C03652=1220.015,344.206,-72.673,-176.049,7.398,148.250
C03653=1220.012,344.454,-72.705,-176.047,7.400,148.250
C03654=1220.007,344.702,-72.737,-176.045,7.403,148.251
C03655=1220.003,344.950,-72.769,-176.043,7.406,148.251
C03656=1219.998,345.198,-72.801,-176.042,7.408,148.251
C03657=1219.994,345.445,-72.833,-176.040,7.412,148.251
C03658=1219.990,345.693,-72.864,-176.038,7.414,148.251
C03659=1219.986,345.942,-72.897,-176.036,7.418,148.252
C03660=1219.982,346.189,-72.928,-176.034,7.420,148.252
C03661=1219.977,346.437,-72.961,-176.032,7.423,148.252
C03662=1219.974,346.685,-72.993,-176.030,7.426,148.252
C03663=1219.969,346.932,-73.025,-176.028,7.428,148.252
C03664=1219.965,347.180,-73.057,-176.027,7.431,148.252
C03665=1219.961,347.429,-73.089,-176.024,7.434,148.253
C03666=1219.956,347.676,-73.121,-176.023,7.437,148.253
C03667=1219.953,347.924,-73.153,-176.021,7.439,148.253
C03668=1219.948,348.173,-73.186,-176.019,7.443,148.253
C03669=1219.945,348.421,-73.217,-176.017,7.445,148.253
C03670=1219.940,348.668,-73.250,-176.015,7.448,148.254
C03671=1219.936,348.916,-73.282,-176.013,7.451,148.254
C03672=1219.932,349.164,-73.314,-176.012,7.453,148.254
C03673=1219.928,349.412,-73.346,-176.010,7.457,148.254
C03674=1219.923,349.660,-73.378,-176.008,7.459,148.254
C03675=1219.919,349.907,-73.411,-176.006,7.462,148.255
C03676=1219.915,350.155,-73.443,-176.004,7.465,148.255
C03677=1219.911,350.403,-73.475,-176.003,7.468,148.255
C03678=1219.906,350.651,-73.507,-176.001,7.471,148.255
C03679=1219.902,350.899,-73.540,-175.999,7.474,148.256
C03680=1219.898,351.147,-73.572,-175.997,7.476,148.256
C03681=1219.894,351.395,-73.605,-175.996,7.479,148.256
C03682=1219.890,351.642,-73.637,-175.994,7.482,148.256
C03683=1219.886,351.890,-73.669,-175.992,7.485,148.256
C03684=1219.882,352.138,-73.701,-175.990,7.488,148.257
C03685=1219.878,352.386,-73.734,-175.988,7.491,148.257
C03686=1219.873,352.634,-73.767,-175.987,7.493,148.257
C03687=1219.869,352.882,-73.798,-175.985,7.497,148.257
C03688=1219.865,353.130,-73.831,-175.983,7.499,148.258
C03689=1219.861,353.378,-73.863,-175.982,7.502,148.258
C03690=1219.857,353.626,-73.896,-175.979,7.505,148.258
C03691=1219.853,353.874,-73.929,-175.978,7.508,148.258
C03692=1219.848,354.121,-73.960,-175.976,7.510,148.258
C03693=1219.844,354.369,-73.993,-175.974,7.514,148.259
C03694=1219.840,354.617,-74.026,-175.973,7.517,148.259
C03695=1219.836,354.864,-74.059,-175.971,7.519,148.259
C03696=1219.832,355.113,-74.091,-175.969,7.522,148.259
C03697=1219.827,355.360,-74.124,-175.967,7.525,148.260
C03698=1219.823,355.608,-74.156,-175.966,7.528,148.260
C03699=1219.819,355.856,-74.188,-175.964,7.530,148.260
C03700=1219.815,356.104,-74.221,-175.962,7.534,148.260
C03701=1219.811,356.352,-74.253,-175.961,7.536,148.261
C03702=1219.807,356.600,-74.286,-175.959,7.539,148.261
C03703=1219.803,356.847,-74.319,-175.957,7.542,148.261
C03704=1219.798,357.095,-74.351,-175.956,7.545,148.261
C03705=1219.794,357.343,-74.384,-175.954,7.547,148.262
C03706=1219.790,357.591,-74.416,-175.952,7.551,148.262
C03707=1219.786,357.839,-74.450,-175.951,7.554,148.262
C03708=1219.782,358.087,-74.481,-175.949,7.556,148.262
C03709=1219.778,358.334,-74.515,-175.948,7.559,148.263
C03710=1219.774,358.582,-74.548,-175.946,7.562,148.263
C03711=1219.769,358.830,-74.580,-175.944,7.565,148.263
C03712=1219.766,359.078,-74.613,-175.943,7.568,148.264
C03713=1219.761,359.326,-74.645,-175.941,7.571,148.264
C03714=1219.757,359.573,-74.678,-175.939,7.574,148.264
C03715=1219.753,359.821,-74.711,-175.938,7.576,148.264
C03716=1219.749,360.069,-74.743,-175.936,7.579,148.265
C03717=1219.745,360.317,-74.776,-175.934,7.582,148.265
C03718=1219.741,360.564,-74.809,-175.933,7.585,148.265
C03719=1219.736,360.813,-74.842,-175.931,7.588,148.265
C03720=1219.732,361.061,-74.875,-175.930,7.590,148.266
C03721=1219.729,361.308,-74.907,-175.928,7.594,148.266
C03722=1219.725,361.556,-74.941,-175.926,7.596,148.266
C03723=1219.720,361.804,-74.973,-175.925,7.599,148.267
C03724=1219.716,362.052,-75.006,-175.923,7.602,148.267
C03725=1219.712,362.300,-75.039,-175.922,7.605,148.267
C03726=1219.708,362.547,-75.072,-175.920,7.608,148.267
C03727=1219.704,362.795,-75.104,-175.919,7.611,148.268
C03728=1219.699,363.042,-75.137,-175.917,7.613,148.268
C03729=1219.695,363.290,-75.170,-175.915,7.617,148.268
C03730=1219.691,363.538,-75.203,-175.914,7.619,148.269
C03731=1219.687,363.785,-75.237,-175.913,7.622,148.269
C03732=1219.682,364.034,-75.269,-175.911,7.625,148.269
C03733=1219.678,364.282,-75.302,-175.909,7.628,148.270
C03734=1219.674,364.529,-75.335,-175.908,7.631,148.270
C03735=1219.670,364.777,-75.368,-175.906,7.634,148.270
C03736=1219.667,365.024,-75.401,-175.905,7.636,148.270
C03737=1219.662,365.272,-75.434,-175.904,7.639,148.271
C03738=1219.658,365.521,-75.467,-175.902,7.643,148.271
C03739=1219.654,365.768,-75.500,-175.900,7.645,148.271
C03740=1219.650,366.016,-75.533,-175.899,7.648,148.272
C03741=1219.646,366.264,-75.566,-175.897,7.651,148.272
C03742=1219.641,366.511,-75.599,-175.896,7.653,148.272
C03743=1219.637,366.791,-75.637,-175.894,7.657,148.273
C03744=1219.633,367.072,-75.674,-175.893,7.660,148.273
C03745=1219.628,367.352,-75.712,-175.891,7.663,148.274
C03746=1219.623,367.631,-75.749,-175.889,7.667,148.274
C03747=1219.619,367.879,-75.782,-175.888,7.670,148.274
C03748=1219.615,368.127,-75.815,-175.887,7.672,148.275
C03749=1219.611,368.374,-75.849,-175.885,7.675,148.275
C03750=1219.607,368.622,-75.882,-175.884,7.678,148.275
C03751=1219.603,368.870,-75.915,-175.883,7.680,148.276
C03752=1219.598,369.117,-75.948,-175.881,7.683,148.276
C03753=1219.594,369.365,-75.981,-175.880,7.686,148.276
C03754=1219.590,369.613,-76.014,-175.878,7.690,148.277
C03755=1219.586,369.861,-76.047,-175.877,7.692,148.277
C03756=1219.582,370.108,-76.081,-175.876,7.695,148.277
C03757=1219.578,370.356,-76.114,-175.874,7.698,148.278
C03758=1219.574,370.604,-76.147,-175.873,7.701,148.278
C03759=1219.569,370.853,-76.181,-175.872,7.703,148.278
C03760=1219.565,371.100,-76.214,-175.870,7.706,148.279
C03761=1219.561,371.348,-76.247,-175.869,7.709,148.279
C03762=1219.557,371.595,-76.281,-175.868,7.712,148.279
C03763=1219.553,371.843,-76.314,-175.867,7.714,148.280
C03764=1219.549,372.091,-76.348,-175.865,7.717,148.280
C03765=1219.545,372.338,-76.381,-175.864,7.720,148.280
C03766=1219.541,372.586,-76.414,-175.863,7.723,148.281
C03767=1219.537,372.834,-76.447,-175.861,7.726,148.281
C03768=1219.532,373.082,-76.480,-175.860,7.729,148.282
C03769=1219.529,373.329,-76.514,-175.859,7.732,148.282
C03770=1219.524,373.577,-76.548,-175.857,7.734,148.282
C03771=1219.520,373.825,-76.581,-175.856,7.737,148.283
C03772=1219.516,374.073,-76.614,-175.855,7.740,148.283
C03773=1219.512,374.321,-76.648,-175.854,7.743,148.283
C03774=1219.508,374.568,-76.681,-175.852,7.746,148.284
C03775=1219.504,374.815,-76.715,-175.851,7.748,148.284
C03776=1219.500,375.063,-76.748,-175.850,7.751,148.285
C03777=1219.495,375.311,-76.782,-175.849,7.754,148.285
C03778=1219.492,375.559,-76.816,-175.848,7.757,148.285
C03779=1219.488,375.807,-76.849,-175.846,7.760,148.286
C03780=1219.483,376.054,-76.882,-175.845,7.763,148.286
C03781=1219.479,376.302,-76.915,-175.844,7.765,148.287
C03782=1219.475,376.549,-76.949,-175.843,7.767,148.287
C03783=1219.471,376.797,-76.983,-175.842,7.770,148.287
C03784=1219.466,377.045,-77.016,-175.841,7.773,148.288
C03785=1219.463,377.293,-77.050,-175.840,7.776,148.288
C03786=1219.459,377.541,-77.083,-175.839,7.779,148.289
C03787=1219.454,377.789,-77.117,-175.838,7.781,148.289
C03788=1219.450,378.036,-77.151,-175.836,7.784,148.289
C03789=1219.446,378.283,-77.184,-175.835,7.787,148.290
C03790=1219.442,378.531,-77.217,-175.834,7.790,148.290
C03791=1219.439,378.779,-77.252,-175.833,7.793,148.291
C03792=1219.434,379.027,-77.285,-175.832,7.796,148.291
C03793=1219.430,379.274,-77.319,-175.830,7.798,148.291
C03794=1219.426,379.522,-77.352,-175.830,7.800,148.292
C03795=1219.422,379.770,-77.386,-175.829,7.803,148.292
C03796=1219.417,380.017,-77.420,-175.827,7.806,148.292
C03797=1219.414,380.265,-77.454,-175.826,7.809,148.293
C03798=1219.410,380.513,-77.487,-175.825,7.812,148.293
C03799=1219.405,380.761,-77.521,-175.824,7.814,148.294
C03800=1219.401,381.008,-77.554,-175.823,7.817,148.294
C03801=1219.397,381.255,-77.588,-175.823,7.820,148.295
C03802=1219.394,381.504,-77.622,-175.821,7.822,148.295
C03803=1219.389,381.751,-77.656,-175.820,7.825,148.295
C03804=1219.385,381.999,-77.689,-175.819,7.828,148.296
C03805=1219.381,382.246,-77.723,-175.818,7.831,148.296
C03806=1219.376,382.494,-77.757,-175.817,7.834,148.297
C03807=1219.373,382.742,-77.791,-175.816,7.836,148.297
C03808=1219.369,382.990,-77.824,-175.815,7.839,148.297
C03809=1219.364,383.237,-77.859,-175.814,7.842,148.298
C03810=1219.360,383.485,-77.892,-175.813,7.844,148.298
C03811=1219.357,383.733,-77.926,-175.812,7.847,148.299
C03812=1219.352,383.981,-77.960,-175.811,7.849,148.299
C03813=1219.348,384.228,-77.994,-175.810,7.852,148.300
C03814=1219.344,384.475,-78.028,-175.809,7.855,148.300
C03815=1219.340,384.724,-78.062,-175.808,7.858,148.300
C03816=1219.336,384.971,-78.096,-175.807,7.860,148.301
C03817=1219.331,385.219,-78.129,-175.806,7.863,148.301
C03818=1219.327,385.466,-78.163,-175.805,7.866,148.302
C03819=1219.324,385.714,-78.197,-175.804,7.869,148.302
C03820=1219.319,385.962,-78.231,-175.804,7.871,148.302
C03821=1219.316,386.209,-78.265,-175.802,7.873,148.303
C03822=1219.311,386.457,-78.299,-175.802,7.877,148.303
C03823=1219.307,386.705,-78.333,-175.801,7.878,148.304
C03824=1219.304,386.952,-78.367,-175.800,7.881,148.304
C03825=1219.299,387.200,-78.401,-175.799,7.884,148.305
C03826=1219.295,387.447,-78.435,-175.798,7.886,148.305
C03827=1219.291,387.696,-78.469,-175.797,7.889,148.306
C03828=1219.287,387.943,-78.503,-175.796,7.892,148.306
C03829=1219.283,388.190,-78.536,-175.796,7.894,148.306
C03830=1219.279,388.438,-78.571,-175.795,7.897,148.307
C03831=1219.275,388.686,-78.604,-175.793,7.900,148.307
C03832=1219.270,388.933,-78.639,-175.793,7.902,148.308
C03833=1219.266,389.180,-78.673,-175.792,7.905,148.308
C03834=1219.262,389.429,-78.707,-175.791,7.908,148.309
C03835=1219.258,389.676,-78.741,-175.790,7.910,148.309
C03836=1219.254,389.924,-78.775,-175.790,7.913,148.310
C03837=1219.250,390.172,-78.809,-175.788,7.916,148.310
C03838=1219.246,390.419,-78.843,-175.788,7.918,148.310
C03839=1219.242,390.667,-78.877,-175.787,7.921,148.311
C03840=1219.239,390.914,-78.911,-175.786,7.923,148.311
C03841=1219.234,391.162,-78.946,-175.785,7.926,148.312
C03842=1219.230,391.410,-78.979,-175.784,7.929,148.312
C03843=1219.226,391.658,-79.014,-175.784,7.931,148.313
C03844=1219.222,391.905,-79.048,-175.783,7.934,148.313
C03845=1219.218,392.152,-79.082,-175.782,7.936,148.314
C03846=1219.214,392.401,-79.116,-175.781,7.939,148.314
C03847=1219.209,392.682,-79.155,-175.780,7.942,148.315
C03848=1219.205,392.964,-79.193,-175.779,7.945,148.315
C03849=1219.200,393.246,-79.233,-175.779,7.948,148.316
C03850=1219.195,393.527,-79.272,-175.778,7.950,148.316
C03851=1219.191,393.775,-79.305,-175.777,7.953,148.316
C03852=1219.187,394.023,-79.340,-175.777,7.955,148.317
C03853=1219.183,394.270,-79.374,-175.776,7.958,148.317
C03854=1219.178,394.518,-79.408,-175.775,7.960,148.318
C03855=1219.175,394.766,-79.443,-175.774,7.963,148.318
C03856=1219.171,395.013,-79.477,-175.774,7.965,148.319
C03857=1219.167,395.260,-79.511,-175.773,7.968,148.319
C03858=1219.163,395.508,-79.546,-175.772,7.970,148.320
C03859=1219.158,395.756,-79.580,-175.771,7.973,148.320
C03860=1219.155,396.004,-79.614,-175.771,7.975,148.320
C03861=1219.150,396.252,-79.648,-175.770,7.978,148.321
C03862=1219.146,396.499,-79.682,-175.769,7.980,148.321
C03863=1219.142,396.747,-79.717,-175.768,7.983,148.322
C03864=1219.138,396.994,-79.751,-175.768,7.985,148.322
C03865=1219.134,397.241,-79.785,-175.767,7.988,148.323
C03866=1219.130,397.489,-79.820,-175.766,7.990,148.323
C03867=1219.126,397.737,-79.854,-175.766,7.992,148.323
C03868=1219.122,397.985,-79.889,-175.765,7.995,148.324
C03869=1219.118,398.232,-79.923,-175.764,7.997,148.324
C03870=1219.114,398.479,-79.957,-175.764,8.000,148.325
C03871=1219.110,398.727,-79.992,-175.763,8.002,148.325
C03872=1219.106,398.974,-80.026,-175.763,8.004,148.326
C03873=1219.101,399.222,-80.060,-175.762,8.007,148.326
C03874=1219.097,399.470,-80.095,-175.761,8.010,148.327
C03875=1219.094,399.717,-80.129,-175.760,8.012,148.327
C03876=1219.090,399.965,-80.164,-175.760,8.014,148.328
C03877=1219.085,400.213,-80.198,-175.759,8.017,148.328
C03878=1219.082,400.460,-80.233,-175.758,8.019,148.329
C03879=1219.077,400.708,-80.267,-175.758,8.022,148.329
C03880=1219.073,400.955,-80.301,-175.757,8.024,148.329
C03881=1219.069,401.203,-80.336,-175.757,8.027,148.330
C03882=1219.065,401.451,-80.370,-175.756,8.029,148.330
C03883=1219.062,401.698,-80.405,-175.756,8.031,148.331
C03884=1219.057,401.946,-80.439,-175.755,8.034,148.331
C03885=1219.052,402.193,-80.473,-175.754,8.036,148.332
C03886=1219.049,402.441,-80.508,-175.754,8.038,148.332
C03887=1219.045,402.688,-80.542,-175.753,8.041,148.333
C03888=1219.041,402.937,-80.577,-175.752,8.043,148.333
C03889=1219.036,403.184,-80.611,-175.752,8.045,148.333
C03890=1219.033,403.432,-80.646,-175.752,8.047,148.334
C03891=1219.028,403.679,-80.680,-175.750,8.050,148.334
C03892=1219.024,403.927,-80.715,-175.750,8.053,148.335
C03893=1219.021,404.174,-80.750,-175.750,8.055,148.335
C03894=1219.016,404.421,-80.784,-175.749,8.058,148.336
C03895=1219.012,404.669,-80.819,-175.748,8.060,148.336
C03896=1219.008,404.917,-80.853,-175.748,8.062,148.337
C03897=1219.005,405.165,-80.888,-175.747,8.064,148.337
C03898=1219.000,405.412,-80.922,-175.747,8.067,148.338
C03899=1218.996,405.660,-80.957,-175.746,8.069,148.338
C03900=1218.992,405.907,-80.992,-175.746,8.071,148.339
C03901=1218.988,406.155,-81.026,-175.745,8.073,148.339
C03902=1218.984,406.402,-81.061,-175.745,8.075,148.339
C03903=1218.980,406.650,-81.096,-175.744,8.078,148.340
C03904=1218.976,406.897,-81.130,-175.744,8.081,148.340
C03905=1218.972,407.145,-81.164,-175.743,8.083,148.341
C03906=1218.968,407.392,-81.200,-175.743,8.085,148.341
C03907=1218.963,407.640,-81.234,-175.742,8.087,148.342
C03908=1218.960,407.888,-81.268,-175.741,8.090,148.342
C03909=1218.956,408.135,-81.303,-175.741,8.092,148.342
C03910=1218.952,408.383,-81.338,-175.740,8.094,148.343
C03911=1218.947,408.630,-81.373,-175.740,8.096,148.343
C03912=1218.944,408.878,-81.407,-175.739,8.098,148.344
C03913=1218.939,409.125,-81.441,-175.738,8.101,148.344
C03914=1218.936,409.373,-81.476,-175.738,8.103,148.345
C03915=1218.931,409.620,-81.511,-175.738,8.105,148.345
C03916=1218.927,409.868,-81.546,-175.737,8.107,148.346
C03917=1218.923,410.115,-81.580,-175.737,8.110,148.346
C03918=1218.919,410.363,-81.615,-175.736,8.112,148.346
C03919=1218.915,410.610,-81.650,-175.736,8.114,148.347
C03920=1218.911,410.858,-81.685,-175.735,8.117,148.347
C03921=1218.907,411.106,-81.719,-175.735,8.119,148.348
C03922=1218.903,411.353,-81.754,-175.734,8.121,148.348
C03923=1218.899,411.600,-81.789,-175.734,8.123,148.349
C03924=1218.895,411.848,-81.824,-175.733,8.125,148.349
C03925=1218.891,412.096,-81.858,-175.732,8.127,148.349
C03926=1218.887,412.343,-81.894,-175.732,8.129,148.350
C03927=1218.883,412.590,-81.928,-175.732,8.131,148.350
C03928=1218.879,412.839,-81.962,-175.731,8.135,148.351
C03929=1218.875,413.085,-81.998,-175.730,8.137,148.351
C03930=1218.871,413.333,-82.032,-175.730,8.139,148.352
C03931=1218.867,413.582,-82.067,-175.729,8.141,148.352
C03932=1218.863,413.828,-82.102,-175.729,8.143,148.353
C03933=1218.859,414.077,-82.137,-175.728,8.145,148.353
C03934=1218.855,414.324,-82.171,-175.728,8.147,148.354
C03935=1218.851,414.571,-82.207,-175.728,8.149,148.354
C03936=1218.847,414.819,-82.241,-175.727,8.151,148.354
C03937=1218.843,415.067,-82.276,-175.727,8.153,148.355
C03938=1218.838,415.313,-82.311,-175.726,8.155,148.355
C03939=1218.836,415.536,-82.343,-175.726,8.158,148.356
C03940=1218.831,415.758,-82.373,-175.725,8.160,148.356
C03941=1218.827,415.980,-82.404,-175.725,8.162,148.356
C03942=1218.825,416.202,-82.436,-175.724,8.164,148.357
C03943=1218.820,416.424,-82.467,-175.724,8.166,148.357
C03944=1218.817,416.647,-82.499,-175.724,8.167,148.357
C03945=1218.814,416.868,-82.530,-175.723,8.169,148.358
C03946=1218.815,417.091,-82.561,-175.723,8.171,148.358
C03947=1218.392,417.091,-82.596,-175.726,8.182,148.362
C03948=1218.392,416.867,-82.564,-175.726,8.180,148.362
C03949=1218.395,416.643,-82.533,-175.727,8.178,148.361
C03950=1218.398,416.421,-82.501,-175.728,8.176,148.361
C03951=1218.402,416.197,-82.470,-175.727,8.174,148.360
C03952=1218.406,415.973,-82.439,-175.728,8.172,148.360
C03953=1218.410,415.750,-82.407,-175.729,8.170,148.360
C03954=1218.414,415.527,-82.376,-175.729,8.168,148.359
C03955=1218.417,415.303,-82.344,-175.730,8.166,148.359
C03956=1218.421,415.056,-82.309,-175.730,8.164,148.358
C03957=1218.425,414.808,-82.275,-175.730,8.162,148.358
C03958=1218.429,414.561,-82.240,-175.731,8.160,148.358
C03959=1218.433,414.313,-82.205,-175.731,8.158,148.357
C03960=1218.437,414.065,-82.170,-175.732,8.156,148.357
C03961=1218.441,413.818,-82.135,-175.732,8.153,148.356
C03962=1218.445,413.570,-82.100,-175.733,8.151,148.356
C03963=1218.449,413.323,-82.065,-175.733,8.149,148.355
C03964=1218.453,413.075,-82.030,-175.734,8.147,148.355
C03965=1218.457,412.828,-81.996,-175.734,8.145,148.354
C03966=1218.461,412.581,-81.961,-175.735,8.142,148.354
C03967=1218.465,412.333,-81.926,-175.735,8.140,148.354
C03968=1218.469,412.085,-81.892,-175.736,8.138,148.353
C03969=1218.474,411.838,-81.857,-175.736,8.136,148.353
C03970=1218.477,411.590,-81.822,-175.737,8.134,148.352
C03971=1218.481,411.343,-81.788,-175.737,8.132,148.352
C03972=1218.485,411.095,-81.753,-175.737,8.129,148.351
C03973=1218.489,410.848,-81.718,-175.738,8.127,148.351
C03974=1218.493,410.600,-81.683,-175.739,8.124,148.350
C03975=1218.498,410.353,-81.648,-175.740,8.122,148.350
C03976=1218.501,410.105,-81.614,-175.740,8.120,148.350
C03977=1218.505,409.858,-81.579,-175.740,8.118,148.349
C03978=1218.509,409.610,-81.544,-175.741,8.116,148.349
C03979=1218.514,409.362,-81.510,-175.741,8.114,148.348
C03980=1218.518,409.114,-81.475,-175.741,8.112,148.348
C03981=1218.521,408.868,-81.440,-175.743,8.109,148.347
C03982=1218.525,408.620,-81.405,-175.743,8.106,148.347
C03983=1218.530,408.372,-81.371,-175.743,8.104,148.347
C03984=1218.534,408.124,-81.336,-175.744,8.102,148.346
C03985=1218.538,407.878,-81.301,-175.744,8.100,148.346
C03986=1218.542,407.629,-81.267,-175.744,8.098,148.345
C03987=1218.546,407.382,-81.232,-175.746,8.095,148.345
C03988=1218.550,407.134,-81.197,-175.746,8.093,148.344
C03989=1218.555,406.887,-81.163,-175.747,8.091,148.344
C03990=1218.558,406.639,-81.128,-175.747,8.089,148.343
C03991=1218.562,406.392,-81.093,-175.747,8.087,148.343
C03992=1218.566,406.144,-81.059,-175.748,8.084,148.342
C03993=1218.571,405.896,-81.024,-175.749,8.082,148.342
C03994=1218.574,405.649,-80.990,-175.749,8.079,148.342
C03995=1218.578,405.401,-80.955,-175.750,8.077,148.341
C03996=1218.583,405.154,-80.920,-175.750,8.074,148.341
C03997=1218.586,404.907,-80.886,-175.751,8.072,148.340
C03998=1218.591,404.659,-80.852,-175.752,8.070,148.340
C03999=1218.594,404.411,-80.817,-175.752,8.068,148.339
C04000=1218.599,404.164,-80.782,-175.753,8.065,148.339
C04001=1218.602,403.916,-80.748,-175.753,8.063,148.338
C04002=1218.607,403.668,-80.714,-175.754,8.061,148.338
C04003=1218.611,403.420,-80.679,-175.754,8.059,148.338
C04004=1218.614,403.174,-80.644,-175.755,8.056,148.337
C04005=1218.618,402.926,-80.609,-175.755,8.054,148.337
C04006=1218.623,402.678,-80.575,-175.756,8.052,148.336
C04007=1218.627,402.431,-80.541,-175.757,8.048,148.336
C04008=1218.631,402.183,-80.506,-175.757,8.046,148.335
C04009=1218.635,401.936,-80.472,-175.758,8.044,148.335
C04010=1218.639,401.687,-80.437,-175.759,8.041,148.334
C04011=1218.643,401.440,-80.403,-175.759,8.039,148.334
C04012=1218.647,401.192,-80.368,-175.760,8.037,148.334
C04013=1218.652,400.945,-80.334,-175.760,8.034,148.333
C04014=1218.655,400.698,-80.300,-175.761,8.032,148.333
C04015=1218.659,400.450,-80.265,-175.761,8.030,148.332
C04016=1218.664,400.202,-80.231,-175.762,8.027,148.332
C04017=1218.667,399.954,-80.196,-175.763,8.025,148.331
C04018=1218.672,399.707,-80.162,-175.763,8.023,148.331
C04019=1218.676,399.460,-80.128,-175.764,8.020,148.330
C04020=1218.680,399.212,-80.093,-175.765,8.018,148.330
C04021=1218.684,398.964,-80.059,-175.766,8.015,148.329
C04022=1218.687,398.716,-80.024,-175.766,8.013,148.329
C04023=1218.692,398.469,-79.990,-175.767,8.011,148.329
C04024=1218.697,398.222,-79.955,-175.767,8.007,148.328
C04025=1218.700,397.974,-79.921,-175.768,8.005,148.328
C04026=1218.704,397.726,-79.887,-175.769,8.002,148.327
C04027=1218.708,397.479,-79.853,-175.769,8.000,148.327
C04028=1218.712,397.231,-79.818,-175.770,7.998,148.326
C04029=1218.717,396.984,-79.784,-175.771,7.995,148.326
C04030=1218.720,396.736,-79.749,-175.771,7.993,148.325
C04031=1218.724,396.488,-79.715,-175.772,7.990,148.325
C04032=1218.728,396.241,-79.681,-175.773,7.988,148.325
C04033=1218.732,395.993,-79.646,-175.774,7.985,148.324
C04034=1218.737,395.746,-79.612,-175.774,7.983,148.324
C04035=1218.740,395.498,-79.577,-175.775,7.980,148.323
C04036=1218.745,395.250,-79.544,-175.776,7.978,148.323
C04037=1218.749,395.003,-79.510,-175.776,7.976,148.322
C04038=1218.753,394.755,-79.475,-175.777,7.973,148.322
C04039=1218.757,394.508,-79.441,-175.778,7.971,148.321
C04040=1218.761,394.260,-79.407,-175.778,7.968,148.321
C04041=1218.765,394.012,-79.372,-175.779,7.966,148.320
C04042=1218.769,393.765,-79.338,-175.780,7.963,148.320
C04043=1218.774,393.518,-79.304,-175.781,7.960,148.319
C04044=1218.777,393.235,-79.265,-175.782,7.958,148.319
C04045=1218.782,392.953,-79.226,-175.782,7.955,148.318
C04046=1218.787,392.671,-79.187,-175.784,7.952,148.318
C04047=1218.792,392.390,-79.148,-175.784,7.949,148.317
C04048=1218.795,392.143,-79.114,-175.785,7.946,148.317
C04049=1218.800,391.894,-79.080,-175.786,7.944,148.317
C04050=1218.804,391.647,-79.046,-175.787,7.941,148.316
C04051=1218.808,391.399,-79.012,-175.787,7.939,148.316
C04052=1218.811,391.152,-78.977,-175.788,7.936,148.315
C04053=1218.816,390.904,-78.943,-175.789,7.933,148.315
C04054=1218.820,390.656,-78.910,-175.790,7.931,148.314
C04055=1218.824,390.408,-78.875,-175.791,7.928,148.314
C04056=1218.828,390.161,-78.841,-175.791,7.926,148.314
C04057=1218.832,389.914,-78.807,-175.792,7.923,148.313
C04058=1218.836,389.665,-78.773,-175.793,7.920,148.313
C04059=1218.841,389.418,-78.739,-175.794,7.918,148.312
C04060=1218.844,389.171,-78.705,-175.795,7.915,148.312
C04061=1218.849,388.923,-78.671,-175.795,7.913,148.311
C04062=1218.852,388.675,-78.637,-175.797,7.910,148.311
C04063=1218.857,388.427,-78.602,-175.797,7.907,148.310
C04064=1218.861,388.180,-78.568,-175.798,7.905,148.310
C04065=1218.864,387.932,-78.535,-175.799,7.902,148.310
C04066=1218.869,387.685,-78.500,-175.800,7.900,148.309
C04067=1218.873,387.437,-78.467,-175.800,7.897,148.309
C04068=1218.878,387.189,-78.433,-175.802,7.894,148.308
C04069=1218.881,386.942,-78.399,-175.803,7.892,148.308
C04070=1218.885,386.694,-78.364,-175.804,7.889,148.307
C04071=1218.890,386.446,-78.331,-175.804,7.887,148.307
C04072=1218.893,386.199,-78.297,-175.805,7.884,148.306
C04073=1218.898,385.951,-78.263,-175.807,7.881,148.306
C04074=1218.902,385.703,-78.229,-175.807,7.879,148.306
C04075=1218.906,385.456,-78.195,-175.808,7.876,148.305
C04076=1218.910,385.208,-78.161,-175.809,7.873,148.305
C04077=1218.913,384.961,-78.127,-175.810,7.870,148.304
C04078=1218.918,384.712,-78.093,-175.811,7.868,148.304
C04079=1218.922,384.465,-78.060,-175.812,7.865,148.303
C04080=1218.925,384.218,-78.025,-175.813,7.862,148.303
C04081=1218.930,383.970,-77.992,-175.814,7.859,148.303
C04082=1218.934,383.722,-77.958,-175.815,7.858,148.302
C04083=1218.938,383.475,-77.925,-175.815,7.854,148.302
C04084=1218.942,383.227,-77.890,-175.817,7.852,148.301
C04085=1218.946,382.979,-77.857,-175.818,7.849,148.301
C04086=1218.950,382.732,-77.823,-175.819,7.846,148.300
C04087=1218.955,382.484,-77.789,-175.820,7.844,148.300
C04088=1218.959,382.237,-77.755,-175.821,7.841,148.300
C04089=1218.962,381.988,-77.722,-175.822,7.838,148.299
C04090=1218.967,381.741,-77.687,-175.823,7.835,148.299
C04091=1218.971,381.493,-77.654,-175.824,7.832,148.298
C04092=1218.975,381.246,-77.620,-175.825,7.830,148.298
C04093=1218.979,380.997,-77.586,-175.826,7.828,148.298
C04094=1218.983,380.750,-77.552,-175.827,7.825,148.297
C04095=1218.987,380.502,-77.519,-175.828,7.822,148.297
C04096=1218.992,380.255,-77.484,-175.829,7.819,148.296
C04097=1218.996,380.007,-77.451,-175.830,7.816,148.296
C04098=1219.000,379.759,-77.418,-175.831,7.813,148.295
C04099=1219.003,379.512,-77.384,-175.832,7.810,148.295
C04100=1219.008,379.264,-77.350,-175.833,7.808,148.295
C04101=1219.012,379.016,-77.316,-175.834,7.806,148.294
C04102=1219.016,378.769,-77.283,-175.835,7.803,148.294
C04103=1219.020,378.521,-77.250,-175.837,7.800,148.294
C04104=1219.024,378.273,-77.215,-175.838,7.797,148.293
C04105=1219.028,378.025,-77.182,-175.839,7.794,148.293
C04106=1219.033,377.777,-77.149,-175.840,7.792,148.292
C04107=1219.036,377.530,-77.115,-175.841,7.789,148.292
C04108=1219.041,377.282,-77.081,-175.843,7.786,148.292
C04109=1219.045,377.035,-77.048,-175.844,7.783,148.291
C04110=1219.049,376.787,-77.014,-175.845,7.780,148.291
C04111=1219.053,376.539,-76.981,-175.846,7.777,148.290
C04112=1219.057,376.291,-76.948,-175.847,7.775,148.290
C04113=1219.061,376.044,-76.913,-175.848,7.772,148.290
C04114=1219.066,375.796,-76.880,-175.850,7.769,148.289
C04115=1219.070,375.548,-76.847,-175.851,7.766,148.289
C04116=1219.074,375.301,-76.813,-175.851,7.764,148.288
C04117=1219.077,375.053,-76.779,-175.853,7.761,148.288
C04118=1219.081,374.805,-76.746,-175.854,7.759,148.288
C04119=1219.086,374.557,-76.712,-175.855,7.756,148.287
C04120=1219.090,374.310,-76.679,-175.856,7.753,148.287
C04121=1219.094,374.062,-76.645,-175.858,7.749,148.286
C04122=1219.098,373.815,-76.612,-175.859,7.746,148.286
C04123=1219.102,373.567,-76.579,-175.861,7.744,148.286
C04124=1219.106,373.319,-76.546,-175.862,7.741,148.285
C04125=1219.110,373.071,-76.512,-175.863,7.738,148.285
C04126=1219.115,372.823,-76.478,-175.864,7.735,148.285
C04127=1219.119,372.575,-76.445,-175.865,7.733,148.284
C04128=1219.123,372.328,-76.412,-175.867,7.730,148.284
C04129=1219.127,372.080,-76.379,-175.868,7.727,148.283
C04130=1219.131,371.832,-76.345,-175.869,7.724,148.283
C04131=1219.135,371.585,-76.312,-175.871,7.722,148.283
C04132=1219.139,371.337,-76.278,-175.872,7.719,148.282
C04133=1219.143,371.090,-76.245,-175.873,7.716,148.282
C04134=1219.147,370.842,-76.212,-175.874,7.713,148.282
C04135=1219.152,370.594,-76.179,-175.876,7.711,148.282
C04136=1219.156,370.347,-76.146,-175.877,7.708,148.281
C04137=1219.159,370.098,-76.112,-175.878,7.705,148.281
C04138=1219.164,369.850,-76.078,-175.880,7.701,148.280
C04139=1219.168,369.602,-76.045,-175.882,7.699,148.280
C04140=1219.172,369.355,-76.012,-175.883,7.696,148.280
C04141=1219.177,369.107,-75.979,-175.884,7.693,148.279
C04142=1219.181,368.859,-75.946,-175.885,7.690,148.279
C04143=1219.185,368.611,-75.913,-175.887,7.688,148.279
C04144=1219.189,368.364,-75.879,-175.888,7.685,148.278
C04145=1219.193,368.116,-75.846,-175.889,7.682,148.278
C04146=1219.197,367.868,-75.813,-175.891,7.679,148.278
C04147=1219.201,367.621,-75.780,-175.893,7.676,148.277
C04148=1219.206,367.341,-75.742,-175.894,7.673,148.277
C04149=1219.211,367.061,-75.705,-175.895,7.670,148.276
C04150=1219.215,366.781,-75.668,-175.897,7.667,148.276
C04151=1219.219,366.501,-75.630,-175.899,7.663,148.276
C04152=1219.224,366.253,-75.597,-175.900,7.661,148.275
C04153=1219.228,366.005,-75.564,-175.902,7.658,148.275
C04154=1219.232,365.758,-75.531,-175.903,7.654,148.275
C04155=1219.236,365.510,-75.498,-175.905,7.652,148.275
C04156=1219.240,365.262,-75.464,-175.906,7.649,148.274
C04157=1219.244,365.014,-75.431,-175.907,7.646,148.274
C04158=1219.249,364.766,-75.399,-175.909,7.644,148.274
C04159=1219.252,364.519,-75.366,-175.911,7.640,148.273
C04160=1219.256,364.271,-75.333,-175.912,7.638,148.273
C04161=1219.260,364.023,-75.300,-175.914,7.635,148.273
C04162=1219.265,363.776,-75.267,-175.915,7.632,148.272
C04163=1219.269,363.528,-75.234,-175.917,7.629,148.272
C04164=1219.273,363.279,-75.201,-175.919,7.626,148.272
C04165=1219.277,363.032,-75.168,-175.920,7.623,148.271
C04166=1219.281,362.784,-75.135,-175.921,7.621,148.271
C04167=1219.285,362.537,-75.102,-175.923,7.618,148.271
C04168=1219.290,362.290,-75.070,-175.925,7.615,148.271
C04169=1219.294,362.041,-75.037,-175.926,7.612,148.270
C04170=1219.298,361.793,-75.004,-175.928,7.609,148.270
C04171=1219.302,361.546,-74.971,-175.929,7.606,148.270
C04172=1219.306,361.298,-74.938,-175.931,7.603,148.269
C04173=1219.311,361.050,-74.905,-175.933,7.600,148.269
C04174=1219.314,360.802,-74.873,-175.934,7.598,148.269
C04175=1219.318,360.554,-74.840,-175.936,7.594,148.269
C04176=1219.323,360.306,-74.807,-175.937,7.591,148.268
C04177=1219.327,360.058,-74.774,-175.939,7.589,148.268
C04178=1219.331,359.811,-74.741,-175.940,7.586,148.268
C04179=1219.335,359.563,-74.709,-175.942,7.583,148.267
C04180=1219.339,359.315,-74.676,-175.944,7.580,148.267
C04181=1219.343,359.067,-74.643,-175.945,7.577,148.267
C04182=1219.348,358.820,-74.611,-175.947,7.574,148.267
C04183=1219.352,358.572,-74.578,-175.949,7.572,148.266
C04184=1219.356,358.324,-74.545,-175.950,7.569,148.266
C04185=1219.360,358.076,-74.512,-175.952,7.566,148.266
C04186=1219.364,357.828,-74.479,-175.954,7.563,148.266
C04187=1219.368,357.580,-74.447,-175.955,7.560,148.265
C04188=1219.372,357.333,-74.414,-175.957,7.558,148.265
C04189=1219.376,357.085,-74.381,-175.959,7.554,148.265
C04190=1219.381,356.836,-74.349,-175.960,7.552,148.265
C04191=1219.385,356.590,-74.316,-175.962,7.549,148.264
C04192=1219.389,356.341,-74.284,-175.964,7.545,148.264
C04193=1219.393,356.094,-74.251,-175.965,7.543,148.264
C04194=1219.397,355.846,-74.219,-175.967,7.540,148.264
C04195=1219.401,355.598,-74.186,-175.969,7.537,148.263
C04196=1219.406,355.350,-74.153,-175.970,7.534,148.263
C04197=1219.409,355.102,-74.121,-175.972,7.532,148.263
C04198=1219.414,354.854,-74.089,-175.974,7.529,148.263
C04199=1219.418,354.607,-74.056,-175.976,7.526,148.262
C04200=1219.422,354.359,-74.024,-175.977,7.523,148.262
C04201=1219.426,354.110,-73.991,-175.979,7.520,148.262
C04202=1219.430,353.863,-73.958,-175.981,7.517,148.262
C04203=1219.435,353.615,-73.927,-175.983,7.515,148.261
C04204=1219.439,353.368,-73.894,-175.984,7.512,148.261
C04205=1219.443,353.119,-73.861,-175.986,7.508,148.261
C04206=1219.447,352.871,-73.829,-175.988,7.506,148.261
C04207=1219.451,352.623,-73.796,-175.990,7.503,148.260
C04208=1219.455,352.376,-73.765,-175.991,7.500,148.260
C04209=1219.460,352.128,-73.732,-175.993,7.498,148.260
C04210=1219.464,351.880,-73.699,-175.995,7.494,148.260
C04211=1219.468,351.632,-73.667,-175.997,7.492,148.260
C04212=1219.472,351.384,-73.635,-175.999,7.489,148.259
C04213=1219.476,351.137,-73.603,-176.001,7.486,148.259
C04214=1219.481,350.889,-73.570,-176.002,7.483,148.259
C04215=1219.484,350.641,-73.538,-176.004,7.480,148.259
C04216=1219.488,350.393,-73.505,-176.006,7.477,148.258
C04217=1219.493,350.145,-73.474,-176.007,7.475,148.258
C04218=1219.497,349.897,-73.441,-176.009,7.472,148.258
C04219=1219.502,349.649,-73.409,-176.011,7.469,148.258
C04220=1219.505,349.401,-73.376,-176.013,7.466,148.258
C04221=1219.510,349.154,-73.344,-176.014,7.464,148.257
C04222=1219.514,348.906,-73.312,-176.017,7.460,148.257
C04223=1219.518,348.657,-73.280,-176.018,7.458,148.257
C04224=1219.522,348.409,-73.248,-176.020,7.454,148.257
C04225=1219.527,348.162,-73.215,-176.022,7.452,148.257
C04226=1219.530,347.914,-73.183,-176.024,7.449,148.256
C04227=1219.534,347.666,-73.151,-176.026,7.446,148.256
C04228=1219.539,347.418,-73.119,-176.028,7.443,148.256
C04229=1219.543,347.170,-73.088,-176.029,7.441,148.256
C04230=1219.547,346.922,-73.055,-176.031,7.438,148.256
C04231=1219.551,346.674,-73.023,-176.033,7.435,148.255
C04232=1219.556,346.427,-72.990,-176.035,7.432,148.255
C04233=1219.559,346.179,-72.959,-176.037,7.429,148.255
C04234=1219.564,345.931,-72.926,-176.039,7.427,148.255
C04235=1219.568,345.683,-72.895,-176.041,7.423,148.255
C04236=1219.572,345.435,-72.863,-176.043,7.421,148.255
C04237=1219.576,345.187,-72.830,-176.045,7.418,148.254
C04238=1219.581,344.940,-72.799,-176.047,7.415,148.254
C04239=1219.585,344.691,-72.767,-176.048,7.413,148.254
C04240=1219.589,344.443,-72.735,-176.050,7.409,148.254
C04241=1219.593,344.196,-72.703,-176.052,7.407,148.254
C04242=1219.598,343.948,-72.671,-176.054,7.404,148.253
C04243=1219.601,343.700,-72.639,-176.056,7.401,148.253
C04244=1219.606,343.452,-72.607,-176.058,7.398,148.253
C04245=1219.610,343.204,-72.575,-176.060,7.395,148.253
C04246=1219.614,342.956,-72.543,-176.062,7.393,148.253
C04247=1219.619,342.708,-72.511,-176.064,7.390,148.253
C04248=1219.622,342.460,-72.479,-176.066,7.387,148.252
C04249=1219.626,342.211,-72.448,-176.067,7.384,148.252
C04250=1219.632,341.964,-72.416,-176.070,7.381,148.252
C04251=1219.635,341.716,-72.384,-176.072,7.379,148.252
C04252=1219.640,341.438,-72.349,-176.074,7.375,148.252
C04253=1219.645,341.160,-72.312,-176.076,7.372,148.252
C04254=1219.649,340.882,-72.277,-176.078,7.369,148.251
C04255=1219.654,340.605,-72.242,-176.080,7.367,148.251
C04256=1219.659,340.357,-72.210,-176.083,7.363,148.251
C04257=1219.662,340.109,-72.178,-176.084,7.361,148.251
C04258=1219.666,339.860,-72.147,-176.086,7.357,148.251
C04259=1219.671,339.613,-72.115,-176.088,7.355,148.251
C04260=1219.675,339.365,-72.083,-176.090,7.353,148.251
C04261=1219.679,339.117,-72.051,-176.092,7.349,148.250
C04262=1219.683,338.869,-72.020,-176.094,7.347,148.250
C04263=1219.688,338.621,-71.989,-176.097,7.344,148.250
C04264=1219.691,338.373,-71.957,-176.098,7.341,148.250
C04265=1219.696,338.125,-71.925,-176.100,7.339,148.250
C04266=1219.700,337.878,-71.893,-176.103,7.336,148.250
C04267=1219.704,337.629,-71.862,-176.104,7.333,148.250
C04268=1219.708,337.382,-71.830,-176.106,7.330,148.249
C04269=1219.712,337.134,-71.799,-176.108,7.327,148.249
C04270=1219.718,336.885,-71.767,-176.111,7.324,148.249
C04271=1219.721,336.637,-71.735,-176.112,7.322,148.249
C04272=1219.726,336.390,-71.704,-176.114,7.319,148.249
C04273=1219.730,336.141,-71.673,-176.117,7.316,148.249
C04274=1219.734,335.894,-71.641,-176.118,7.313,148.249
C04275=1219.738,335.646,-71.609,-176.121,7.310,148.249
C04276=1219.742,335.398,-71.579,-176.122,7.308,148.248
C04277=1219.746,335.150,-71.547,-176.124,7.305,148.248
C04278=1219.751,334.902,-71.515,-176.127,7.302,148.248
C04279=1219.755,334.654,-71.484,-176.128,7.300,148.248
C04280=1219.760,334.406,-71.453,-176.131,7.296,148.248
C04281=1219.763,334.158,-71.421,-176.133,7.294,148.248
C04282=1219.768,333.910,-71.390,-176.135,7.291,148.248
C04283=1219.772,333.662,-71.358,-176.137,7.289,148.248
C04284=1219.776,333.414,-71.327,-176.139,7.286,148.248
C04285=1219.780,333.166,-71.296,-176.141,7.283,148.247
C04286=1219.784,332.918,-71.264,-176.143,7.281,148.247
C04287=1219.788,332.670,-71.233,-176.145,7.277,148.247
C04288=1219.793,332.422,-71.202,-176.147,7.275,148.247
C04289=1219.797,332.174,-71.171,-176.149,7.272,148.247
C04290=1219.801,331.926,-71.140,-176.152,7.269,148.247
C04291=1219.805,331.678,-71.108,-176.153,7.267,148.247
C04292=1219.809,331.430,-71.077,-176.156,7.264,148.247
C04293=1219.813,331.182,-71.045,-176.157,7.261,148.247
C04294=1219.818,330.934,-71.015,-176.160,7.258,148.247
C04295=1219.822,330.686,-70.983,-176.162,7.256,148.246
C04296=1219.826,330.438,-70.952,-176.164,7.253,148.246
C04297=1219.831,330.190,-70.921,-176.166,7.250,148.246
C04298=1219.834,329.942,-70.889,-176.168,7.248,148.246
C04299=1219.839,329.694,-70.859,-176.170,7.245,148.246
C04300=1219.843,329.445,-70.827,-176.172,7.242,148.246
C04301=1219.847,329.198,-70.796,-176.175,7.239,148.246
C04302=1219.852,328.950,-70.765,-176.177,7.237,148.246
C04303=1219.856,328.701,-70.734,-176.179,7.233,148.246
C04304=1219.860,328.454,-70.703,-176.181,7.231,148.246
C04305=1219.864,328.205,-70.672,-176.183,7.229,148.246
C04306=1219.869,327.957,-70.641,-176.185,7.226,148.246
C04307=1219.874,327.709,-70.610,-176.187,7.223,148.245
C04308=1219.877,327.461,-70.579,-176.190,7.220,148.245
C04309=1219.881,327.213,-70.548,-176.191,7.218,148.245
C04310=1219.886,326.966,-70.517,-176.194,7.214,148.245
C04311=1219.890,326.717,-70.486,-176.196,7.212,148.245
C04312=1219.894,326.469,-70.455,-176.198,7.209,148.245
C04313=1219.899,326.222,-70.424,-176.200,7.207,148.245
C04314=1219.903,325.973,-70.393,-176.202,7.204,148.245
C04315=1219.907,325.725,-70.363,-176.205,7.201,148.245
C04316=1219.911,325.477,-70.331,-176.207,7.199,148.245
C04317=1219.915,325.229,-70.301,-176.209,7.196,148.245
C04318=1219.920,324.981,-70.270,-176.211,7.193,148.245
C04319=1219.924,324.733,-70.238,-176.213,7.190,148.245
C04320=1219.927,324.485,-70.208,-176.215,7.188,148.245
C04321=1219.932,324.237,-70.177,-176.218,7.186,148.245
C04322=1219.936,323.988,-70.146,-176.220,7.182,148.244
C04323=1219.941,323.740,-70.115,-176.222,7.180,148.245
C04324=1219.945,323.493,-70.085,-176.224,7.177,148.245
C04325=1219.949,323.245,-70.054,-176.226,7.174,148.244
C04326=1219.953,322.996,-70.023,-176.229,7.171,148.244
C04327=1219.958,322.748,-69.992,-176.231,7.169,148.244
C04328=1219.962,322.501,-69.962,-176.233,7.167,148.244
C04329=1219.966,322.252,-69.931,-176.235,7.164,148.244
C04330=1219.970,322.004,-69.900,-176.237,7.161,148.244
C04331=1219.975,321.756,-69.870,-176.239,7.158,148.244
C04332=1219.978,321.508,-69.839,-176.242,7.156,148.244
C04333=1219.983,321.260,-69.808,-176.244,7.153,148.244
C04334=1219.987,321.012,-69.777,-176.246,7.150,148.244
C04335=1219.991,320.764,-69.747,-176.248,7.148,148.244
C04336=1219.995,320.515,-69.716,-176.251,7.145,148.244
C04337=1220.000,320.267,-69.685,-176.253,7.143,148.244
C04338=1220.004,320.020,-69.655,-176.255,7.139,148.244
C04339=1220.008,319.772,-69.624,-176.257,7.137,148.244
C04340=1220.013,319.523,-69.594,-176.260,7.134,148.244
C04341=1220.017,319.275,-69.564,-176.262,7.132,148.244
C04342=1220.021,319.027,-69.533,-176.263,7.129,148.244
C04343=1220.026,318.779,-69.502,-176.266,7.126,148.244
C04344=1220.030,318.531,-69.472,-176.268,7.124,148.244
C04345=1220.034,318.283,-69.441,-176.271,7.121,148.244
C04346=1220.038,318.034,-69.412,-176.273,7.119,148.244
C04347=1220.042,317.786,-69.381,-176.275,7.115,148.244
C04348=1220.047,317.539,-69.350,-176.277,7.113,148.244
C04349=1220.051,317.291,-69.320,-176.280,7.110,148.244
C04350=1220.055,317.042,-69.289,-176.282,7.108,148.244
C04351=1220.059,316.794,-69.259,-176.284,7.105,148.244
C04352=1220.064,316.546,-69.229,-176.286,7.102,148.244
C04353=1220.068,316.298,-69.198,-176.288,7.100,148.244
C04354=1220.072,316.050,-69.168,-176.291,7.097,148.244
C04355=1220.077,315.801,-69.137,-176.293,7.095,148.244
C04356=1220.081,315.526,-69.104,-176.296,7.092,148.244
C04357=1220.086,315.250,-69.070,-176.299,7.089,148.244
C04358=1220.091,314.974,-69.036,-176.300,7.086,148.243
C04359=1220.095,314.698,-69.003,-176.303,7.083,148.243
C04360=1220.100,314.450,-68.972,-176.306,7.080,148.243
C04361=1220.104,314.202,-68.942,-176.308,7.078,148.244
C04362=1220.108,313.953,-68.912,-176.310,7.075,148.244
C04363=1220.112,313.705,-68.882,-176.312,7.073,148.244
C04364=1220.117,313.457,-68.852,-176.315,7.070,148.244
C04365=1220.121,313.209,-68.821,-176.317,7.067,148.244
C04366=1220.125,312.962,-68.791,-176.319,7.065,148.243
C04367=1220.130,312.713,-68.761,-176.322,7.062,148.243
C04368=1220.134,312.465,-68.731,-176.324,7.060,148.244
C04369=1220.138,312.217,-68.701,-176.326,7.057,148.244
C04370=1220.142,311.969,-68.671,-176.328,7.054,148.244
C04371=1220.147,311.720,-68.640,-176.331,7.052,148.244
C04372=1220.151,311.472,-68.610,-176.333,7.049,148.244
C04373=1220.155,311.224,-68.581,-176.335,7.047,148.244
C04374=1220.159,310.976,-68.550,-176.338,7.044,148.244
C04375=1220.164,310.728,-68.521,-176.340,7.042,148.244
C04376=1220.168,310.480,-68.490,-176.342,7.039,148.244
C04377=1220.172,310.232,-68.460,-176.344,7.036,148.244
C04378=1220.176,309.984,-68.430,-176.346,7.034,148.244
C04379=1220.181,309.735,-68.400,-176.349,7.031,148.244
C04380=1220.185,309.487,-68.371,-176.351,7.029,148.244
C04381=1220.189,309.239,-68.340,-176.353,7.026,148.244
C04382=1220.194,308.991,-68.310,-176.356,7.023,148.244
C04383=1220.198,308.743,-68.281,-176.358,7.021,148.244
C04384=1220.202,308.495,-68.251,-176.361,7.018,148.244
C04385=1220.207,308.246,-68.221,-176.363,7.016,148.244
C04386=1220.211,307.999,-68.191,-176.366,7.013,148.244
C04387=1220.215,307.750,-68.161,-176.368,7.011,148.244
C04388=1220.220,307.502,-68.131,-176.370,7.008,148.244
C04389=1220.224,307.254,-68.102,-176.372,7.005,148.244
C04390=1220.228,307.006,-68.071,-176.375,7.003,148.244
C04391=1220.232,306.758,-68.042,-176.377,7.000,148.244
C04392=1220.237,306.509,-68.012,-176.379,6.998,148.244
C04393=1220.241,306.261,-67.982,-176.381,6.996,148.244
C04394=1220.245,306.013,-67.952,-176.384,6.993,148.244
C04395=1220.249,305.765,-67.923,-176.386,6.990,148.244
C04396=1220.254,305.516,-67.893,-176.389,6.987,148.244
C04397=1220.259,305.268,-67.863,-176.391,6.985,148.244
C04398=1220.262,305.020,-67.833,-176.393,6.983,148.244
C04399=1220.267,304.772,-67.804,-176.396,6.980,148.244
C04400=1220.272,304.524,-67.774,-176.398,6.978,148.244
C04401=1220.276,304.275,-67.744,-176.401,6.975,148.244
C04402=1220.280,304.027,-67.715,-176.403,6.972,148.244
C04403=1220.284,303.779,-67.685,-176.405,6.970,148.245
C04404=1220.288,303.531,-67.655,-176.407,6.967,148.245
C04405=1220.292,303.283,-67.626,-176.410,6.965,148.245
C04406=1220.297,303.034,-67.596,-176.412,6.962,148.245
C04407=1220.301,302.786,-67.566,-176.414,6.960,148.245
C04408=1220.305,302.538,-67.537,-176.417,6.957,148.245
C04409=1220.310,302.289,-67.507,-176.420,6.955,148.245
C04410=1220.314,302.041,-67.478,-176.422,6.953,148.245
C04411=1220.319,301.794,-67.449,-176.424,6.950,148.245
C04412=1220.323,301.545,-67.419,-176.427,6.947,148.245
C04413=1220.327,301.297,-67.390,-176.429,6.945,148.245
C04414=1220.332,301.048,-67.360,-176.431,6.942,148.245
C04415=1220.336,300.800,-67.330,-176.433,6.940,148.245
C04416=1220.340,300.552,-67.301,-176.436,6.938,148.245
C04417=1220.344,300.304,-67.271,-176.438,6.935,148.245
C04418=1220.349,300.055,-67.242,-176.440,6.932,148.245
C04419=1220.353,299.807,-67.213,-176.443,6.930,148.246
C04420=1220.357,299.559,-67.183,-176.446,6.927,148.246
C04421=1220.362,299.311,-67.154,-176.448,6.925,148.246
C04422=1220.366,299.063,-67.125,-176.450,6.922,148.246
C04423=1220.370,298.815,-67.095,-176.452,6.920,148.246
C04424=1220.374,298.567,-67.066,-176.455,6.918,148.246
C04425=1220.378,298.318,-67.036,-176.457,6.915,148.246
C04426=1220.383,298.069,-67.007,-176.459,6.912,148.246
C04427=1220.388,297.822,-66.978,-176.463,6.910,148.246
C04428=1220.392,297.574,-66.949,-176.465,6.908,148.246
C04429=1220.396,297.325,-66.919,-176.467,6.905,148.246
C04430=1220.400,297.077,-66.890,-176.469,6.902,148.246
C04431=1220.404,296.829,-66.861,-176.472,6.900,148.246
C04432=1220.409,296.580,-66.832,-176.474,6.898,148.246
C04433=1220.414,296.332,-66.803,-176.476,6.895,148.246
C04434=1220.418,296.084,-66.773,-176.479,6.893,148.247
C04435=1220.422,295.836,-66.744,-176.481,6.891,148.247
C04436=1220.427,295.587,-66.715,-176.484,6.888,148.247
C04437=1220.431,295.339,-66.686,-176.486,6.885,148.247
C04438=1220.434,295.091,-66.657,-176.488,6.882,148.247
C04439=1220.439,294.843,-66.628,-176.491,6.881,148.247
C04440=1220.443,294.594,-66.599,-176.493,6.878,148.247
C04441=1220.448,294.346,-66.570,-176.496,6.875,148.247
C04442=1220.452,294.098,-66.540,-176.498,6.873,148.247
C04443=1220.457,293.849,-66.512,-176.500,6.871,148.247
C04444=1220.461,293.601,-66.482,-176.503,6.868,148.247
C04445=1220.465,293.353,-66.453,-176.505,6.866,148.248
C04446=1220.469,293.104,-66.425,-176.507,6.864,148.248
C04447=1220.474,292.857,-66.396,-176.510,6.861,148.248
C04448=1220.478,292.609,-66.366,-176.512,6.858,148.248
C04449=1220.482,292.360,-66.337,-176.515,6.857,148.248
C04450=1220.487,292.111,-66.308,-176.518,6.853,148.248
C04451=1220.492,291.863,-66.280,-176.520,6.851,148.248
C04452=1220.495,291.615,-66.251,-176.522,6.849,148.248
C04453=1220.500,291.366,-66.222,-176.525,6.846,148.248
C04454=1220.504,291.118,-66.192,-176.527,6.844,148.248
C04455=1220.509,290.870,-66.163,-176.529,6.842,148.248
C04456=1220.512,290.622,-66.135,-176.532,6.839,148.248
C04457=1220.517,290.374,-66.106,-176.534,6.837,148.249
C04458=1220.522,290.125,-66.077,-176.537,6.835,148.249
C04459=1220.526,289.877,-66.048,-176.539,6.832,148.249
C04460=1220.531,289.603,-66.016,-176.542,6.830,148.249
C04461=1220.535,289.328,-65.985,-176.544,6.827,148.249
C04462=1220.540,289.054,-65.953,-176.547,6.824,148.249
C04463=1220.545,288.780,-65.921,-176.550,6.822,148.249
C04464=1220.549,288.533,-65.893,-176.552,6.819,148.249
C04465=1220.554,288.284,-65.864,-176.555,6.817,148.250
C04466=1220.558,288.035,-65.835,-176.557,6.815,148.250
C04467=1220.563,287.787,-65.806,-176.560,6.812,148.250
C04468=1220.566,287.539,-65.777,-176.562,6.809,148.250
C04469=1220.571,287.290,-65.749,-176.565,6.808,148.250
C04470=1220.576,287.042,-65.720,-176.567,6.805,148.250
C04471=1220.579,286.794,-65.692,-176.569,6.802,148.250
C04472=1220.584,286.545,-65.663,-176.571,6.800,148.250
C04473=1220.589,286.297,-65.634,-176.575,6.797,148.251
C04474=1220.592,286.049,-65.606,-176.577,6.795,148.251
C04475=1220.597,285.801,-65.577,-176.579,6.793,148.251
C04476=1220.601,285.552,-65.549,-176.582,6.790,148.251
C04477=1220.606,285.303,-65.520,-176.584,6.788,148.251
C04478=1220.610,285.056,-65.491,-176.586,6.786,148.251
C04479=1220.614,284.807,-65.463,-176.589,6.784,148.251
C04480=1220.619,284.558,-65.434,-176.591,6.781,148.251
C04481=1220.623,284.311,-65.407,-176.594,6.779,148.251
C04482=1220.627,284.062,-65.377,-176.596,6.777,148.252
C04483=1220.632,283.814,-65.349,-176.599,6.774,148.252
C04484=1220.636,283.566,-65.321,-176.601,6.772,148.252
C04485=1220.641,283.317,-65.292,-176.604,6.770,148.252
C04486=1220.645,283.069,-65.264,-176.606,6.767,148.252
C04487=1220.649,282.820,-65.235,-176.608,6.764,148.252
C04488=1220.653,282.573,-65.207,-176.611,6.763,148.253
C04489=1220.658,282.324,-65.178,-176.613,6.760,148.253
C04490=1220.662,282.076,-65.150,-176.616,6.758,148.253
C04491=1220.667,281.827,-65.122,-176.618,6.755,148.253
C04492=1220.671,281.579,-65.094,-176.620,6.753,148.253
C04493=1220.676,281.330,-65.065,-176.624,6.750,148.253
C04494=1220.680,281.082,-65.037,-176.626,6.748,148.253
C04495=1220.684,280.833,-65.009,-176.628,6.746,148.253
C04496=1220.689,280.586,-64.981,-176.630,6.744,148.254
C04497=1220.693,280.337,-64.952,-176.633,6.741,148.254
C04498=1220.697,280.088,-64.924,-176.636,6.739,148.254
C04499=1220.702,279.840,-64.896,-176.638,6.737,148.254
C04500=1220.706,279.591,-64.867,-176.641,6.734,148.254
C04501=1220.710,279.344,-64.840,-176.643,6.732,148.254
C04502=1220.715,279.095,-64.811,-176.645,6.730,148.254
C04503=1220.719,278.847,-64.783,-176.648,6.728,148.255
C04504=1220.724,278.598,-64.754,-176.651,6.725,148.255
C04505=1220.728,278.350,-64.727,-176.653,6.723,148.255
C04506=1220.732,278.102,-64.699,-176.655,6.721,148.255
C04507=1220.737,277.853,-64.670,-176.657,6.719,148.255
C04508=1220.741,277.605,-64.642,-176.661,6.716,148.255
C04509=1220.746,277.356,-64.614,-176.663,6.714,148.255
C04510=1220.750,277.109,-64.586,-176.665,6.712,148.256
C04511=1220.754,276.860,-64.558,-176.668,6.709,148.256
C04512=1220.759,276.612,-64.529,-176.670,6.707,148.256
C04513=1220.763,276.363,-64.502,-176.673,6.705,148.256
C04514=1220.767,276.115,-64.474,-176.675,6.703,148.256
C04515=1220.772,275.866,-64.445,-176.678,6.700,148.256
C04516=1220.776,275.618,-64.418,-176.680,6.698,148.257
C04517=1220.780,275.369,-64.389,-176.683,6.696,148.257
C04518=1220.784,275.122,-64.362,-176.685,6.694,148.257
C04519=1220.789,274.873,-64.334,-176.688,6.691,148.257
C04520=1220.793,274.624,-64.306,-176.690,6.689,148.257
C04521=1220.798,274.376,-64.278,-176.692,6.686,148.257
C04522=1220.802,274.127,-64.249,-176.695,6.685,148.258
C04523=1220.807,273.879,-64.222,-176.697,6.681,148.258
C04524=1220.811,273.631,-64.194,-176.700,6.680,148.258
C04525=1220.815,273.382,-64.166,-176.702,6.677,148.258
C04526=1220.820,273.134,-64.139,-176.705,6.676,148.258
C04527=1220.824,272.885,-64.111,-176.707,6.673,148.258
C04528=1220.828,272.637,-64.083,-176.710,6.671,148.259
C04529=1220.833,272.389,-64.056,-176.712,6.668,148.259
C04530=1220.837,272.140,-64.028,-176.715,6.666,148.259
C04531=1220.842,271.892,-63.999,-176.717,6.664,148.259
C04532=1220.846,271.643,-63.972,-176.720,6.662,148.259
C04533=1220.850,271.395,-63.944,-176.722,6.659,148.259
C04534=1220.855,271.147,-63.916,-176.725,6.657,148.260
C04535=1220.859,270.898,-63.889,-176.727,6.655,148.260
C04536=1220.864,270.650,-63.860,-176.730,6.653,148.260
C04537=1220.868,270.401,-63.833,-176.732,6.650,148.260
C04538=1220.873,270.153,-63.806,-176.735,6.648,148.260
C04539=1220.876,269.905,-63.777,-176.737,6.646,148.260
C04540=1220.881,269.656,-63.750,-176.740,6.644,148.261
C04541=1220.885,269.408,-63.723,-176.742,6.641,148.261
C04542=1220.890,269.159,-63.695,-176.745,6.639,148.261
C04543=1220.895,268.911,-63.667,-176.747,6.637,148.261
C04544=1220.899,268.662,-63.640,-176.750,6.635,148.261
C04545=1220.903,268.414,-63.612,-176.752,6.633,148.262
C04546=1220.908,268.165,-63.585,-176.755,6.630,148.262
C04547=1220.912,267.917,-63.557,-176.757,6.628,148.262
C04548=1220.916,267.668,-63.529,-176.760,6.626,148.262
C04549=1220.921,267.420,-63.502,-176.762,6.624,148.262
C04550=1220.925,267.172,-63.474,-176.764,6.622,148.263
C04551=1220.930,266.923,-63.447,-176.767,6.619,148.263
C04552=1220.933,266.675,-63.419,-176.770,6.617,148.263
C04553=1220.938,266.426,-63.392,-176.772,6.615,148.263
C04554=1220.943,266.178,-63.365,-176.774,6.613,148.263
C04555=1220.947,265.930,-63.337,-176.777,6.611,148.264
C04556=1220.951,265.681,-63.310,-176.780,6.608,148.264
C04557=1220.956,265.433,-63.282,-176.782,6.606,148.264
C04558=1220.960,265.184,-63.255,-176.784,6.604,148.264
C04559=1220.965,264.936,-63.228,-176.787,6.602,148.264
C04560=1220.969,264.687,-63.200,-176.789,6.600,148.264
C04561=1220.973,264.439,-63.173,-176.792,6.598,148.265
C04562=1220.978,264.190,-63.146,-176.795,6.596,148.265
C04563=1220.983,263.942,-63.119,-176.797,6.593,148.265
C04564=1220.988,263.669,-63.088,-176.800,6.592,148.265
C04565=1220.992,263.396,-63.058,-176.803,6.589,148.266
C04566=1220.997,263.124,-63.028,-176.805,6.587,148.266
C04567=1221.002,262.851,-62.998,-176.808,6.584,148.266
C04568=1221.006,262.603,-62.971,-176.811,6.582,148.266
C04569=1221.011,262.354,-62.944,-176.813,6.580,148.266
C04570=1221.016,262.106,-62.917,-176.815,6.578,148.267
C04571=1221.019,261.857,-62.889,-176.818,6.575,148.267
C04572=1221.024,261.609,-62.862,-176.821,6.573,148.267
C04573=1221.029,261.360,-62.835,-176.823,6.571,148.267
C04574=1221.033,261.112,-62.808,-176.825,6.569,148.267
C04575=1221.037,260.864,-62.781,-176.828,6.567,148.268
C04576=1221.042,260.615,-62.754,-176.830,6.565,148.268
C04577=1221.046,260.366,-62.727,-176.833,6.563,148.268
C04578=1221.050,260.118,-62.699,-176.836,6.560,148.268
C04579=1221.055,259.869,-62.672,-176.838,6.558,148.268
C04580=1221.060,259.621,-62.645,-176.841,6.556,148.269
C04581=1221.063,259.373,-62.618,-176.843,6.554,148.269
C04582=1221.068,259.124,-62.591,-176.845,6.552,148.269
C04583=1221.073,258.876,-62.564,-176.848,6.550,148.269
C04584=1221.077,258.627,-62.537,-176.851,6.547,148.269
C04585=1221.082,258.378,-62.510,-176.853,6.545,148.270
C04586=1221.085,258.130,-62.483,-176.856,6.543,148.270
C04587=1221.090,257.881,-62.456,-176.858,6.541,148.270
C04588=1221.095,257.633,-62.429,-176.861,6.539,148.270
C04589=1221.099,257.384,-62.402,-176.863,6.537,148.270
C04590=1221.104,257.136,-62.375,-176.865,6.535,148.271
C04591=1221.108,256.888,-62.349,-176.868,6.533,148.271
C04592=1221.113,256.639,-62.322,-176.871,6.530,148.271
C04593=1221.117,256.391,-62.295,-176.873,6.529,148.271
C04594=1221.121,256.142,-62.267,-176.876,6.527,148.272
C04595=1221.125,255.893,-62.241,-176.878,6.524,148.272
C04596=1221.130,255.645,-62.214,-176.881,6.523,148.272
C04597=1221.135,255.396,-62.187,-176.883,6.521,148.272
C04598=1221.139,255.148,-62.161,-176.885,6.519,148.272
C04599=1221.143,254.899,-62.134,-176.888,6.517,148.273
C04600=1221.148,254.651,-62.107,-176.891,6.514,148.273
C04601=1221.152,254.402,-62.080,-176.893,6.512,148.273
C04602=1221.157,254.154,-62.053,-176.896,6.510,148.273
C04603=1221.161,253.905,-62.026,-176.899,6.508,148.274
C04604=1221.166,253.657,-62.000,-176.901,6.506,148.274
C04605=1221.170,253.408,-61.973,-176.903,6.504,148.274
C04606=1221.175,253.160,-61.946,-176.906,6.502,148.274
C04607=1221.179,252.911,-61.920,-176.908,6.500,148.274
C04608=1221.183,252.663,-61.893,-176.911,6.497,148.275
C04609=1221.188,252.414,-61.866,-176.914,6.495,148.275
C04610=1221.192,252.166,-61.840,-176.916,6.493,148.275
C04611=1221.197,251.917,-61.813,-176.919,6.491,148.275
C04612=1221.201,251.668,-61.787,-176.921,6.489,148.276
C04613=1221.206,251.420,-61.760,-176.923,6.487,148.276
C04614=1221.211,251.171,-61.733,-176.926,6.485,148.276
C04615=1221.214,250.923,-61.706,-176.929,6.483,148.276
C04616=1221.219,250.674,-61.680,-176.931,6.481,148.277
C04617=1221.223,250.426,-61.654,-176.933,6.479,148.277
C04618=1221.228,250.177,-61.627,-176.936,6.477,148.277
C04619=1221.232,249.929,-61.601,-176.939,6.474,148.277
C04620=1221.237,249.680,-61.574,-176.941,6.473,148.278
C04621=1221.241,249.431,-61.548,-176.944,6.471,148.278
C04622=1221.246,249.183,-61.521,-176.946,6.469,148.278
C04623=1221.250,248.935,-61.494,-176.949,6.467,148.278
C04624=1221.255,248.685,-61.468,-176.951,6.465,148.279
C04625=1221.259,248.437,-61.442,-176.954,6.463,148.279
C04626=1221.264,248.188,-61.415,-176.956,6.461,148.279
C04627=1221.267,247.940,-61.389,-176.959,6.459,148.279
C04628=1221.272,247.691,-61.363,-176.961,6.457,148.280
C04629=1221.277,247.443,-61.336,-176.964,6.455,148.280
C04630=1221.282,247.195,-61.309,-176.966,6.453,148.280
C04631=1221.286,246.946,-61.284,-176.969,6.450,148.280
C04632=1221.290,246.698,-61.257,-176.972,6.448,148.281
C04633=1221.295,246.449,-61.231,-176.974,6.446,148.281
C04634=1221.299,246.200,-61.204,-176.976,6.444,148.281
C04635=1221.304,245.951,-61.178,-176.979,6.442,148.281
C04636=1221.308,245.703,-61.152,-176.982,6.440,148.282
C04637=1221.312,245.454,-61.125,-176.984,6.438,148.282
C04638=1221.317,245.205,-61.099,-176.986,6.436,148.282
C04639=1221.322,244.958,-61.073,-176.989,6.434,148.282
C04640=1221.326,244.709,-61.047,-176.992,6.433,148.283
C04641=1221.330,244.461,-61.020,-176.994,6.430,148.283
C04642=1221.335,244.211,-60.994,-176.996,6.429,148.283
C04643=1221.339,243.963,-60.968,-176.999,6.427,148.283
C04644=1221.343,243.714,-60.942,-177.002,6.425,148.284
C04645=1221.348,243.465,-60.916,-177.004,6.423,148.284
C04646=1221.353,243.217,-60.890,-177.006,6.421,148.284
C04647=1221.358,242.969,-60.863,-177.010,6.418,148.284
C04648=1221.362,242.720,-60.837,-177.012,6.416,148.285
C04649=1221.366,242.471,-60.812,-177.014,6.414,148.285
C04650=1221.370,242.223,-60.785,-177.017,6.412,148.285
C04651=1221.375,241.974,-60.759,-177.020,6.410,148.285
C04652=1221.380,241.726,-60.733,-177.022,6.408,148.286
C04653=1221.384,241.477,-60.708,-177.024,6.406,148.286
C04654=1221.389,241.228,-60.681,-177.027,6.404,148.286
C04655=1221.393,240.980,-60.655,-177.030,6.402,148.286
C04656=1221.397,240.731,-60.629,-177.032,6.401,148.287
C04657=1221.403,240.482,-60.603,-177.035,6.399,148.287
C04658=1221.407,240.234,-60.577,-177.037,6.397,148.287
C04659=1221.411,239.985,-60.551,-177.040,6.395,148.287
C04660=1221.415,239.737,-60.525,-177.042,6.393,148.288
C04661=1221.419,239.488,-60.499,-177.045,6.391,148.288
C04662=1221.425,239.239,-60.473,-177.047,6.389,148.288
C04663=1221.429,238.991,-60.447,-177.050,6.387,148.288
C04664=1221.433,238.742,-60.421,-177.052,6.385,148.289
C04665=1221.437,238.494,-60.395,-177.055,6.383,148.289
C04666=1221.443,238.245,-60.370,-177.057,6.381,148.289
C04667=1221.447,237.996,-60.344,-177.060,6.379,148.290
C04668=1221.452,237.724,-60.316,-177.062,6.377,148.290
C04669=1221.457,237.454,-60.287,-177.065,6.375,148.290
C04670=1221.461,237.182,-60.259,-177.068,6.373,148.290
C04671=1221.467,236.911,-60.232,-177.071,6.371,148.291
C04672=1221.471,236.662,-60.206,-177.073,6.369,148.291
C04673=1221.475,236.413,-60.180,-177.076,6.367,148.291
C04674=1221.479,236.165,-60.154,-177.078,6.365,148.292
C04675=1221.485,235.917,-60.128,-177.081,6.363,148.292
C04676=1221.489,235.668,-60.102,-177.083,6.361,148.292
C04677=1221.493,235.419,-60.076,-177.086,6.359,148.292
C04678=1221.498,235.171,-60.051,-177.088,6.357,148.293
C04679=1221.502,234.922,-60.025,-177.091,6.356,148.293
C04680=1221.507,234.673,-60.000,-177.094,6.354,148.293
C04681=1221.511,234.424,-59.974,-177.096,6.351,148.293
C04682=1221.516,234.176,-59.949,-177.098,6.350,148.294
C04683=1221.520,233.927,-59.923,-177.101,6.348,148.294
C04684=1221.524,233.678,-59.897,-177.104,6.346,148.294
C04685=1221.530,233.430,-59.871,-177.106,6.344,148.295
C04686=1221.534,233.181,-59.846,-177.109,6.342,148.295
C04687=1221.538,232.932,-59.820,-177.111,6.340,148.295
C04688=1221.543,232.684,-59.794,-177.114,6.338,148.295
C04689=1221.547,232.435,-59.769,-177.116,6.336,148.296
C04690=1221.552,232.186,-59.744,-177.119,6.334,148.296
C04691=1221.557,231.938,-59.718,-177.122,6.333,148.296
C04692=1221.561,231.689,-59.693,-177.124,6.331,148.297
C04693=1221.566,231.441,-59.667,-177.127,6.329,148.297
C04694=1221.570,231.192,-59.641,-177.129,6.327,148.297
C04695=1221.574,230.943,-59.616,-177.132,6.325,148.298
C04696=1221.579,230.694,-59.591,-177.134,6.323,148.298
C04697=1221.583,230.446,-59.565,-177.137,6.321,148.298
C04698=1221.588,230.197,-59.540,-177.140,6.319,148.298
C04699=1221.592,229.949,-59.514,-177.142,6.317,148.299
C04700=1221.596,229.700,-59.490,-177.145,6.315,148.299
C04701=1221.601,229.452,-59.464,-177.147,6.313,148.299
C04702=1221.605,229.203,-59.439,-177.150,6.311,148.300
C04703=1221.610,228.954,-59.413,-177.152,6.309,148.300
C04704=1221.615,228.705,-59.388,-177.155,6.308,148.300
C04705=1221.619,228.456,-59.362,-177.157,6.306,148.301
C04706=1221.624,228.208,-59.337,-177.160,6.304,148.301
C04707=1221.628,227.959,-59.312,-177.163,6.302,148.301
C04708=1221.633,227.711,-59.287,-177.165,6.300,148.301
C04709=1221.637,227.462,-59.261,-177.167,6.298,148.302
C04710=1221.642,227.213,-59.236,-177.170,6.296,148.302
C04711=1221.646,226.965,-59.211,-177.173,6.294,148.302
C04712=1221.650,226.715,-59.186,-177.175,6.292,148.303
C04713=1221.655,226.467,-59.161,-177.178,6.291,148.303
C04714=1221.659,226.218,-59.135,-177.181,6.289,148.303
C04715=1221.665,225.970,-59.110,-177.183,6.287,148.304
C04716=1221.669,225.721,-59.084,-177.186,6.285,148.304
C04717=1221.673,225.472,-59.060,-177.188,6.283,148.304
C04718=1221.677,225.224,-59.035,-177.191,6.281,148.304
C04719=1221.683,224.975,-59.010,-177.193,6.280,148.305
C04720=1221.687,224.726,-58.984,-177.195,6.278,148.305
C04721=1221.692,224.478,-58.959,-177.198,6.276,148.305
C04722=1221.695,224.229,-58.934,-177.201,6.274,148.306
C04723=1221.700,223.981,-58.909,-177.203,6.272,148.306
C04724=1221.705,223.731,-58.884,-177.206,6.271,148.306
C04725=1221.710,223.483,-58.859,-177.208,6.269,148.307
C04726=1221.714,223.234,-58.833,-177.211,6.267,148.307
C04727=1221.719,222.985,-58.809,-177.214,6.265,148.307
C04728=1221.723,222.737,-58.784,-177.216,6.263,148.308
C04729=1221.728,222.488,-58.759,-177.218,6.261,148.308
C04730=1221.732,222.239,-58.733,-177.221,6.259,148.308
C04731=1221.737,221.991,-58.709,-177.224,6.257,148.308
C04732=1221.741,221.741,-58.684,-177.226,6.255,148.309
C04733=1221.746,221.493,-58.659,-177.229,6.254,148.309
C04734=1221.750,221.244,-58.634,-177.232,6.252,148.309
C04735=1221.754,220.996,-58.609,-177.234,6.250,148.310
C04736=1221.760,220.747,-58.584,-177.237,6.248,148.310
C04737=1221.763,220.498,-58.560,-177.239,6.247,148.310
C04738=1221.768,220.250,-58.534,-177.242,6.245,148.311
C04739=1221.773,220.001,-58.509,-177.244,6.243,148.311
C04740=1221.777,219.752,-58.485,-177.247,6.241,148.311
C04741=1221.781,219.503,-58.460,-177.249,6.240,148.312
C04742=1221.787,219.255,-58.435,-177.252,6.238,148.312
C04743=1221.791,219.006,-58.411,-177.255,6.236,148.312
C04744=1221.795,218.757,-58.386,-177.257,6.234,148.313
C04745=1221.800,218.509,-58.360,-177.260,6.232,148.313
C04746=1221.804,218.260,-58.336,-177.263,6.230,148.313
C04747=1221.809,218.011,-58.311,-177.265,6.228,148.313
C04748=1221.814,217.762,-58.287,-177.267,6.226,148.314
C04749=1221.818,217.514,-58.261,-177.270,6.224,148.314
C04750=1221.823,217.265,-58.237,-177.273,6.223,148.314
C04751=1221.827,217.016,-58.212,-177.275,6.221,148.315
C04752=1221.832,216.767,-58.188,-177.277,6.220,148.315
C04753=1221.836,216.519,-58.164,-177.280,6.218,148.315
C04754=1221.841,216.269,-58.139,-177.283,6.216,148.316
C04755=1221.845,216.021,-58.114,-177.285,6.214,148.316
C04756=1221.850,215.773,-58.089,-177.288,6.212,148.316
C04757=1221.854,215.524,-58.065,-177.291,6.210,148.317
C04758=1221.859,215.275,-58.040,-177.293,6.209,148.317
C04759=1221.863,215.026,-58.016,-177.296,6.207,148.317
C04760=1221.868,214.777,-57.991,-177.298,6.205,148.318
C04761=1221.872,214.529,-57.967,-177.301,6.203,148.318
C04762=1221.877,214.280,-57.942,-177.304,6.201,148.318
C04763=1221.881,214.031,-57.918,-177.306,6.200,148.319
C04764=1221.886,213.782,-57.893,-177.308,6.198,148.319
C04765=1221.891,213.534,-57.869,-177.311,6.196,148.319
C04766=1221.895,213.284,-57.844,-177.314,6.195,148.320
C04767=1221.900,213.036,-57.820,-177.316,6.193,148.320
C04768=1221.905,212.787,-57.795,-177.319,6.191,148.320
C04769=1221.909,212.539,-57.771,-177.322,6.189,148.321
C04770=1221.914,212.289,-57.746,-177.324,6.187,148.321
C04771=1221.918,212.041,-57.722,-177.327,6.185,148.321
C04772=1221.923,211.771,-57.695,-177.329,6.183,148.322
C04773=1221.928,211.500,-57.668,-177.332,6.182,148.322
C04774=1221.933,211.230,-57.642,-177.335,6.180,148.323
C04775=1221.938,210.959,-57.616,-177.338,6.178,148.323
C04776=1221.943,210.710,-57.591,-177.340,6.176,148.323
C04777=1221.947,210.462,-57.567,-177.343,6.174,148.324
C04778=1221.952,210.213,-57.542,-177.346,6.173,148.324
C04779=1221.956,209.964,-57.518,-177.348,6.171,148.324
C04780=1221.960,209.716,-57.494,-177.351,6.169,148.325
C04781=1221.966,209.467,-57.470,-177.353,6.168,148.325
C04782=1221.969,209.218,-57.445,-177.356,6.166,148.325
C04783=1221.974,208.969,-57.422,-177.358,6.164,148.326
C04784=1221.979,208.720,-57.397,-177.361,6.162,148.326
C04785=1221.984,208.472,-57.373,-177.364,6.160,148.326
C04786=1221.987,208.223,-57.349,-177.366,6.159,148.327
C04787=1221.993,207.974,-57.324,-177.369,6.157,148.327
C04788=1221.997,207.725,-57.300,-177.372,6.155,148.327
C04789=1222.002,207.476,-57.276,-177.374,6.154,148.328
C04790=1222.007,207.228,-57.252,-177.376,6.152,148.328
C04791=1222.011,206.979,-57.227,-177.379,6.150,148.328
C04792=1222.015,206.730,-57.204,-177.382,6.148,148.329
C04793=1222.020,206.481,-57.180,-177.384,6.147,148.329
C04794=1222.025,206.232,-57.155,-177.387,6.145,148.329
C04795=1222.029,205.984,-57.131,-177.389,6.143,148.330
C04796=1222.034,205.735,-57.108,-177.392,6.142,148.330
C04797=1222.038,205.486,-57.083,-177.394,6.140,148.330
C04798=1222.043,205.237,-57.059,-177.397,6.138,148.331
C04799=1222.048,204.988,-57.035,-177.400,6.137,148.331
C04800=1222.052,204.740,-57.011,-177.403,6.135,148.332
C04801=1222.056,204.491,-56.987,-177.405,6.133,148.332
C04802=1222.062,204.242,-56.963,-177.407,6.132,148.332
C04803=1222.066,203.993,-56.939,-177.410,6.130,148.333
C04804=1222.070,203.744,-56.915,-177.413,6.128,148.333
C04805=1222.075,203.495,-56.891,-177.415,6.126,148.333
C04806=1222.079,203.247,-56.867,-177.418,6.124,148.334
C04807=1222.084,202.998,-56.844,-177.420,6.123,148.334
C04808=1222.089,202.749,-56.819,-177.423,6.122,148.335
C04809=1222.094,202.500,-56.796,-177.425,6.120,148.335
C04810=1222.098,202.252,-56.772,-177.428,6.118,148.335
C04811=1222.102,202.003,-56.747,-177.430,6.116,148.336
C04812=1222.106,201.754,-56.724,-177.433,6.114,148.336
C04813=1222.111,201.505,-56.700,-177.436,6.112,148.336
C04814=1222.116,201.256,-56.677,-177.438,6.111,148.337
C04815=1222.121,201.008,-56.652,-177.441,6.110,148.337
C04816=1222.125,200.758,-56.629,-177.444,6.108,148.337
C04817=1222.130,200.510,-56.604,-177.446,6.106,148.338
C04818=1222.134,200.261,-56.581,-177.449,6.104,148.338
C04819=1222.139,200.013,-56.557,-177.451,6.103,148.339
C04820=1222.144,199.764,-56.534,-177.454,6.101,148.339
C04821=1222.148,199.515,-56.510,-177.456,6.100,148.339
C04822=1222.153,199.266,-56.486,-177.459,6.098,148.340
C04823=1222.157,199.017,-56.463,-177.462,6.096,148.340
C04824=1222.161,198.768,-56.438,-177.464,6.095,148.340
C04825=1222.166,198.519,-56.415,-177.466,6.093,148.341
C04826=1222.171,198.270,-56.392,-177.469,6.091,148.341
C04827=1222.175,198.022,-56.368,-177.472,6.089,148.341
C04828=1222.180,197.772,-56.344,-177.475,6.088,148.342
C04829=1222.184,197.524,-56.320,-177.477,6.087,148.342
C04830=1222.189,197.275,-56.297,-177.479,6.085,148.343
C04831=1222.193,197.026,-56.273,-177.482,6.083,148.343
C04832=1222.198,196.777,-56.250,-177.485,6.081,148.343
C04833=1222.203,196.529,-56.226,-177.487,6.080,148.344
C04834=1222.207,196.280,-56.203,-177.489,6.078,148.344
C04835=1222.212,196.031,-56.179,-177.492,6.077,148.344
C04836=1222.216,195.782,-56.155,-177.495,6.075,148.345
C04837=1222.221,195.533,-56.132,-177.497,6.073,148.345
C04838=1222.226,195.284,-56.109,-177.500,6.071,148.346
C04839=1222.230,195.035,-56.085,-177.503,6.070,148.346
C04840=1222.235,194.787,-56.061,-177.505,6.069,148.346
C04841=1222.240,194.538,-56.038,-177.508,6.067,148.347
C04842=1222.244,194.289,-56.014,-177.510,6.065,148.347
C04843=1222.249,194.039,-55.991,-177.513,6.064,148.347
C04844=1222.254,193.790,-55.968,-177.515,6.062,148.348
C04845=1222.259,193.543,-55.944,-177.518,6.060,148.348
C04846=1222.263,193.294,-55.921,-177.521,6.059,148.349
C04847=1222.268,193.045,-55.897,-177.524,6.057,148.349
C04848=1222.272,192.796,-55.874,-177.526,6.056,148.349
C04849=1222.277,192.547,-55.851,-177.528,6.054,148.350
C04850=1222.281,192.298,-55.828,-177.531,6.052,148.350
C04851=1222.286,192.049,-55.804,-177.534,6.050,148.350
C04852=1222.290,191.800,-55.780,-177.536,6.049,148.351
C04853=1222.295,191.551,-55.757,-177.538,6.048,148.351
C04854=1222.300,191.302,-55.734,-177.542,6.046,148.352
C04855=1222.304,191.054,-55.711,-177.544,6.044,148.352
C04856=1222.309,190.805,-55.687,-177.546,6.043,148.352
C04857=1222.313,190.556,-55.664,-177.549,6.041,148.353
C04858=1222.319,190.307,-55.641,-177.552,6.039,148.353
C04859=1222.323,190.058,-55.618,-177.554,6.038,148.353
C04860=1222.328,189.809,-55.594,-177.556,6.037,148.354
C04861=1222.332,189.560,-55.572,-177.559,6.035,148.354
C04862=1222.337,189.311,-55.548,-177.562,6.033,148.355
C04863=1222.341,189.062,-55.525,-177.565,6.031,148.355
C04864=1222.346,188.813,-55.502,-177.567,6.030,148.356
C04865=1222.350,188.565,-55.479,-177.569,6.029,148.356
C04866=1222.355,188.316,-55.455,-177.572,6.027,148.356
C04867=1222.360,188.067,-55.432,-177.574,6.026,148.357
C04868=1222.365,187.818,-55.409,-177.577,6.024,148.357
C04869=1222.369,187.570,-55.386,-177.580,6.022,148.358
C04870=1222.373,187.321,-55.363,-177.583,6.021,148.358
C04871=1222.378,187.071,-55.340,-177.585,6.020,148.358
C04872=1222.383,186.822,-55.316,-177.587,6.018,148.359
C04873=1222.387,186.574,-55.294,-177.590,6.016,148.359
C04874=1222.392,186.325,-55.271,-177.593,6.014,148.360
C04875=1222.397,186.076,-55.248,-177.595,6.013,148.360
C04876=1222.402,185.806,-55.223,-177.598,6.012,148.360
C04877=1222.407,185.537,-55.198,-177.600,6.010,148.361
C04878=1222.412,185.267,-55.173,-177.604,6.008,148.361
C04879=1222.416,184.998,-55.148,-177.606,6.006,148.362
C04880=1222.421,184.748,-55.126,-177.609,6.005,148.362
C04881=1222.426,184.499,-55.102,-177.611,6.004,148.362
C04882=1222.430,184.251,-55.079,-177.614,6.002,148.363
C04883=1222.435,184.002,-55.056,-177.617,6.000,148.363
C04884=1222.439,183.753,-55.034,-177.619,5.998,148.364
C04885=1222.444,183.504,-55.011,-177.622,5.997,148.364
C04886=1222.449,183.255,-54.988,-177.624,5.996,148.364
C04887=1222.453,183.006,-54.965,-177.627,5.994,148.365
C04888=1222.458,182.758,-54.942,-177.629,5.993,148.365
C04889=1222.463,182.508,-54.920,-177.632,5.991,148.366
C04890=1222.467,182.259,-54.897,-177.635,5.989,148.366
C04891=1222.472,182.010,-54.873,-177.637,5.988,148.366
C04892=1222.477,181.762,-54.851,-177.639,5.987,148.367
C04893=1222.482,181.513,-54.828,-177.643,5.985,148.367
C04894=1222.486,181.264,-54.805,-177.645,5.983,148.368
C04895=1222.491,181.014,-54.783,-177.647,5.982,148.368
C04896=1222.495,180.766,-54.760,-177.650,5.980,148.368
C04897=1222.500,180.517,-54.737,-177.653,5.979,148.369
C04898=1222.504,180.268,-54.715,-177.655,5.978,148.369
C04899=1222.509,180.019,-54.692,-177.658,5.976,148.370
C04900=1222.514,179.771,-54.669,-177.661,5.974,148.370
C04901=1222.518,179.521,-54.647,-177.663,5.973,148.370
C04902=1222.523,179.272,-54.623,-177.666,5.972,148.371
C04903=1222.528,179.024,-54.601,-177.668,5.970,148.371
C04904=1222.533,178.774,-54.578,-177.671,5.969,148.372
C04905=1222.537,178.525,-54.556,-177.673,5.967,148.372
C04906=1222.541,178.277,-54.534,-177.676,5.965,148.372
C04907=1222.546,178.028,-54.510,-177.678,5.965,148.373
C04908=1222.550,177.779,-54.488,-177.681,5.963,148.373
C04909=1222.555,177.530,-54.465,-177.684,5.961,148.374
C04910=1222.560,177.281,-54.443,-177.686,5.960,148.374
C04911=1222.565,177.032,-54.420,-177.688,5.958,148.374
C04912=1222.569,176.783,-54.398,-177.692,5.957,148.375
C04913=1222.574,176.534,-54.375,-177.694,5.956,148.375
C04914=1222.579,176.285,-54.353,-177.696,5.954,148.376
C04915=1222.583,176.036,-54.331,-177.699,5.952,148.376
C04916=1222.588,175.787,-54.308,-177.702,5.951,148.377
C04917=1222.592,175.538,-54.286,-177.704,5.949,148.377
C04918=1222.598,175.290,-54.263,-177.707,5.948,148.377
C04919=1222.602,175.040,-54.241,-177.709,5.947,148.378
C04920=1222.606,174.792,-54.218,-177.712,5.945,148.378
C04921=1222.612,174.543,-54.196,-177.715,5.943,148.379
C04922=1222.616,174.293,-54.174,-177.717,5.942,148.379
C04923=1222.621,174.044,-54.150,-177.720,5.940,148.380
C04924=1222.625,173.796,-54.129,-177.722,5.939,148.380
C04925=1222.630,173.546,-54.106,-177.725,5.938,148.381
C04926=1222.635,173.298,-54.083,-177.727,5.936,148.381
C04927=1222.639,173.049,-54.061,-177.729,5.935,148.381
C04928=1222.643,172.799,-54.039,-177.732,5.933,148.382
C04929=1222.649,172.551,-54.016,-177.735,5.932,148.382
C04930=1222.653,172.302,-53.994,-177.737,5.931,148.383
C04931=1222.658,172.053,-53.973,-177.740,5.929,148.383
C04932=1222.662,171.804,-53.950,-177.743,5.927,148.383
C04933=1222.667,171.555,-53.928,-177.745,5.926,148.384
C04934=1222.672,171.306,-53.906,-177.748,5.925,148.384
C04935=1222.676,171.057,-53.884,-177.750,5.924,148.385
C04936=1222.681,170.808,-53.861,-177.753,5.922,148.385
C04937=1222.686,170.559,-53.838,-177.756,5.920,148.386
C04938=1222.690,170.310,-53.817,-177.758,5.919,148.386
C04939=1222.695,170.061,-53.795,-177.761,5.917,148.386
C04940=1222.700,169.813,-53.772,-177.764,5.916,148.387
C04941=1222.704,169.563,-53.750,-177.766,5.915,148.387
C04942=1222.709,169.315,-53.728,-177.768,5.913,148.388
C04943=1222.713,169.065,-53.706,-177.771,5.912,148.388
C04944=1222.719,168.816,-53.684,-177.774,5.911,148.389
C04945=1222.723,168.567,-53.662,-177.776,5.909,148.389
C04946=1222.727,168.318,-53.639,-177.778,5.908,148.389
C04947=1222.732,168.070,-53.617,-177.781,5.906,148.390
C04948=1222.736,167.820,-53.595,-177.784,5.905,148.390
C04949=1222.742,167.571,-53.573,-177.786,5.904,148.391
C04950=1222.746,167.322,-53.551,-177.789,5.902,148.391
C04951=1222.751,167.073,-53.529,-177.792,5.901,148.392
C04952=1222.755,166.824,-53.507,-177.794,5.899,148.392
C04953=1222.760,166.575,-53.485,-177.796,5.898,148.393
C04954=1222.765,166.326,-53.463,-177.799,5.896,148.393
C04955=1222.769,166.077,-53.442,-177.802,5.895,148.393
C04956=1222.774,165.828,-53.419,-177.804,5.894,148.394
C04957=1222.779,165.579,-53.397,-177.807,5.892,148.394
C04958=1222.784,165.331,-53.376,-177.810,5.891,148.395
C04959=1222.788,165.082,-53.353,-177.812,5.890,148.395
C04960=1222.793,164.833,-53.331,-177.814,5.889,148.396
C04961=1222.798,164.583,-53.310,-177.817,5.887,148.396
C04962=1222.802,164.335,-53.288,-177.820,5.885,148.397
C04963=1222.807,164.085,-53.266,-177.822,5.884,148.397
C04964=1222.812,163.837,-53.244,-177.825,5.883,148.397
C04965=1222.816,163.587,-53.222,-177.827,5.882,148.398
C04966=1222.821,163.338,-53.200,-177.830,5.880,148.398
C04967=1222.826,163.090,-53.178,-177.833,5.878,148.399
C04968=1222.831,162.840,-53.156,-177.835,5.878,148.399
C04969=1222.835,162.592,-53.135,-177.838,5.876,148.400
C04970=1222.840,162.342,-53.113,-177.840,5.875,148.400
C04971=1222.845,162.094,-53.091,-177.843,5.873,148.401
C04972=1222.849,161.844,-53.069,-177.845,5.872,148.401
C04973=1222.854,161.596,-53.047,-177.848,5.870,148.401
C04974=1222.859,161.346,-53.026,-177.851,5.870,148.402
C04975=1222.863,161.097,-53.004,-177.853,5.868,148.402
C04976=1222.868,160.848,-52.983,-177.856,5.866,148.403
C04977=1222.872,160.599,-52.961,-177.858,5.865,148.403
C04978=1222.877,160.350,-52.939,-177.861,5.864,148.404
C04979=1222.882,160.102,-52.917,-177.863,5.863,148.404
C04980=1222.887,159.833,-52.894,-177.866,5.861,148.405
C04981=1222.892,159.563,-52.871,-177.869,5.859,148.405
C04982=1222.897,159.295,-52.847,-177.872,5.858,148.406
C04983=1222.902,159.026,-52.824,-177.874,5.857,148.406
C04984=1222.906,158.776,-52.802,-177.877,5.855,148.407
C04985=1222.911,158.528,-52.780,-177.880,5.854,148.407
C04986=1222.916,158.278,-52.759,-177.882,5.853,148.407
C04987=1222.921,158.029,-52.737,-177.885,5.852,148.408
C04988=1222.926,157.780,-52.716,-177.888,5.850,148.408
C04989=1222.930,157.530,-52.694,-177.890,5.848,148.409
C04990=1222.935,157.282,-52.673,-177.893,5.848,148.409
C04991=1222.940,157.033,-52.651,-177.895,5.846,148.410
C04992=1222.944,156.783,-52.630,-177.898,5.845,148.410
C04993=1222.949,156.535,-52.609,-177.901,5.843,148.411
C04994=1222.954,156.286,-52.587,-177.903,5.842,148.411
C04995=1222.959,156.037,-52.566,-177.905,5.841,148.411
C04996=1222.963,155.788,-52.544,-177.908,5.840,148.412
C04997=1222.968,155.539,-52.522,-177.911,5.838,148.412
C04998=1222.973,155.290,-52.501,-177.913,5.837,148.413
C04999=1222.977,155.040,-52.479,-177.916,5.836,148.413
C05000=1222.981,154.792,-52.458,-177.918,5.835,148.414
C05001=1222.987,154.543,-52.437,-177.921,5.833,148.414
C05002=1222.991,154.293,-52.415,-177.923,5.832,148.415
C05003=1222.996,154.044,-52.394,-177.926,5.830,148.415
C05004=1223.001,153.796,-52.373,-177.928,5.829,148.416
C05005=1223.005,153.547,-52.352,-177.931,5.828,148.416
C05006=1223.010,153.297,-52.330,-177.933,5.827,148.417
C05007=1223.014,153.049,-52.308,-177.937,5.825,148.417
C05008=1223.020,152.799,-52.287,-177.939,5.824,148.418
C05009=1223.025,152.551,-52.266,-177.941,5.823,148.418
C05010=1223.028,152.301,-52.245,-177.944,5.822,148.419
C05011=1223.033,152.052,-52.223,-177.947,5.820,148.419
C05012=1223.038,151.803,-52.202,-177.949,5.819,148.419
C05013=1223.044,151.554,-52.181,-177.952,5.818,148.420
C05014=1223.048,151.306,-52.160,-177.954,5.817,148.420
C05015=1223.052,151.056,-52.139,-177.957,5.815,148.421
C05016=1223.057,150.807,-52.117,-177.959,5.814,148.421
C05017=1223.062,150.558,-52.096,-177.962,5.812,148.422
C05018=1223.066,150.309,-52.075,-177.964,5.812,148.422
C05019=1223.071,150.059,-52.054,-177.967,5.810,148.423
C05020=1223.076,149.811,-52.032,-177.969,5.809,148.423
C05021=1223.080,149.562,-52.012,-177.972,5.808,148.424
C05022=1223.086,149.313,-51.991,-177.974,5.807,148.424
C05023=1223.090,149.064,-51.969,-177.978,5.805,148.425
C05024=1223.094,148.814,-51.948,-177.980,5.804,148.425
C05025=1223.099,148.565,-51.928,-177.982,5.802,148.426
C05026=1223.104,148.316,-51.906,-177.985,5.802,148.426
C05027=1223.109,148.067,-51.885,-177.988,5.800,148.427
C05028=1223.114,147.818,-51.864,-177.990,5.799,148.427
C05029=1223.119,147.570,-51.843,-177.993,5.797,148.428
C05030=1223.123,147.320,-51.822,-177.995,5.796,148.428
C05031=1223.128,147.071,-51.801,-177.998,5.795,148.429
C05032=1223.133,146.822,-51.779,-178.000,5.794,148.429
C05033=1223.137,146.573,-51.759,-178.003,5.793,148.430
C05034=1223.142,146.324,-51.738,-178.006,5.792,148.430
C05035=1223.147,146.075,-51.718,-178.008,5.790,148.430
C05036=1223.152,145.826,-51.696,-178.011,5.789,148.431
C05037=1223.156,145.576,-51.675,-178.013,5.787,148.431
C05038=1223.161,145.327,-51.654,-178.016,5.787,148.432
C05039=1223.166,145.078,-51.633,-178.018,5.786,148.432
C05040=1223.170,144.830,-51.612,-178.021,5.784,148.433
C05041=1223.175,144.580,-51.591,-178.023,5.783,148.433
C05042=1223.179,144.331,-51.571,-178.026,5.781,148.434
C05043=1223.185,144.082,-51.550,-178.029,5.781,148.434
C05044=1223.190,143.833,-51.529,-178.031,5.779,148.435
C05045=1223.193,143.584,-51.508,-178.034,5.778,148.435
C05046=1223.199,143.335,-51.487,-178.037,5.776,148.436
C05047=1223.203,143.086,-51.466,-178.039,5.775,148.436
C05048=1223.208,142.836,-51.445,-178.042,5.774,148.437
C05049=1223.213,142.588,-51.425,-178.044,5.773,148.437
C05050=1223.218,142.338,-51.404,-178.047,5.772,148.438
C05051=1223.222,142.089,-51.384,-178.049,5.771,148.438
C05052=1223.227,141.840,-51.363,-178.052,5.770,148.439
C05053=1223.232,141.591,-51.342,-178.055,5.768,148.439
C05054=1223.237,141.342,-51.320,-178.057,5.767,148.440
C05055=1223.241,141.094,-51.300,-178.060,5.766,148.440
C05056=1223.246,140.844,-51.279,-178.062,5.765,148.441
C05057=1223.251,140.595,-51.259,-178.065,5.764,148.441
C05058=1223.255,140.346,-51.238,-178.067,5.762,148.442
C05059=1223.260,140.096,-51.217,-178.070,5.762,148.442
C05060=1223.264,139.847,-51.197,-178.072,5.760,148.443
C05061=1223.269,139.598,-51.176,-178.075,5.759,148.443
C05062=1223.274,139.349,-51.155,-178.078,5.757,148.444
C05063=1223.279,139.100,-51.134,-178.080,5.756,148.444
C05064=1223.283,138.851,-51.114,-178.082,5.756,148.445
C05065=1223.288,138.602,-51.094,-178.085,5.754,148.445
C05066=1223.293,138.353,-51.073,-178.088,5.753,148.446
C05067=1223.297,138.104,-51.052,-178.090,5.752,148.446
C05068=1223.303,137.855,-51.031,-178.093,5.751,148.447
C05069=1223.307,137.606,-51.011,-178.096,5.749,148.447
C05070=1223.312,137.356,-50.991,-178.098,5.748,148.448
C05071=1223.317,137.107,-50.970,-178.100,5.747,148.448
C05072=1223.321,136.858,-50.950,-178.104,5.746,148.449
C05073=1223.326,136.609,-50.930,-178.106,5.745,148.449
C05074=1223.331,136.360,-50.909,-178.109,5.744,148.450
C05075=1223.335,136.111,-50.888,-178.111,5.743,148.450
C05076=1223.340,135.862,-50.868,-178.113,5.742,148.450
C05077=1223.345,135.613,-50.847,-178.116,5.740,148.451
C05078=1223.350,135.364,-50.827,-178.118,5.739,148.451
C05079=1223.354,135.114,-50.807,-178.122,5.738,148.452
C05080=1223.360,134.865,-50.786,-178.124,5.737,148.452
C05081=1223.364,134.617,-50.766,-178.126,5.736,148.453
C05082=1223.369,134.368,-50.746,-178.129,5.734,148.453
C05083=1223.374,134.118,-50.725,-178.131,5.734,148.454
C05084=1223.378,133.849,-50.703,-178.134,5.732,148.455
C05085=1223.384,133.581,-50.681,-178.137,5.731,148.455
C05086=1223.389,133.312,-50.659,-178.140,5.730,148.456
C05087=1223.394,133.044,-50.637,-178.143,5.728,148.456
C05088=1223.399,132.794,-50.617,-178.145,5.727,148.457
C05089=1223.404,132.545,-50.597,-178.147,5.726,148.457
C05090=1223.408,132.296,-50.576,-178.150,5.725,148.458
C05091=1223.413,132.047,-50.556,-178.153,5.724,148.458
C05092=1223.418,131.797,-50.536,-178.155,5.723,148.459
C05093=1223.423,131.548,-50.515,-178.158,5.722,148.459
C05094=1223.428,131.300,-50.495,-178.160,5.721,148.460
C05095=1223.433,131.050,-50.476,-178.163,5.719,148.460
C05096=1223.437,130.801,-50.455,-178.166,5.718,148.461
C05097=1223.442,130.552,-50.434,-178.168,5.717,148.461
C05098=1223.447,130.302,-50.415,-178.171,5.716,148.462
C05099=1223.451,130.054,-50.394,-178.173,5.715,148.462
C05100=1223.456,129.805,-50.374,-178.176,5.714,148.463
C05101=1223.460,129.555,-50.354,-178.178,5.713,148.463
C05102=1223.466,129.307,-50.334,-178.181,5.712,148.464
C05103=1223.471,129.057,-50.313,-178.184,5.710,148.464
C05104=1223.475,128.808,-50.294,-178.186,5.710,148.465
C05105=1223.480,128.559,-50.273,-178.188,5.709,148.465
C05106=1223.485,128.309,-50.254,-178.192,5.707,148.466
C05107=1223.489,128.060,-50.233,-178.194,5.706,148.466
C05108=1223.494,127.811,-50.214,-178.196,5.706,148.467
C05109=1223.499,127.563,-50.194,-178.199,5.704,148.467
C05110=1223.504,127.313,-50.173,-178.202,5.703,148.468
C05111=1223.509,127.064,-50.153,-178.204,5.702,148.468
C05112=1223.513,126.815,-50.133,-178.207,5.701,148.469
C05113=1223.518,126.565,-50.113,-178.209,5.700,148.469
C05114=1223.522,126.316,-50.093,-178.212,5.699,148.470
C05115=1223.528,126.067,-50.073,-178.215,5.698,148.471
C05116=1223.532,125.819,-50.053,-178.217,5.697,148.471
C05117=1223.537,125.569,-50.033,-178.220,5.695,148.472
C05118=1223.541,125.320,-50.013,-178.222,5.694,148.472
C05119=1223.546,125.070,-49.993,-178.225,5.694,148.473
C05120=1223.551,124.822,-49.974,-178.227,5.692,148.473
C05121=1223.556,124.573,-49.953,-178.230,5.691,148.474
C05122=1223.561,124.323,-49.934,-178.232,5.690,148.474
C05123=1223.565,124.074,-49.913,-178.235,5.689,148.475
C05124=1223.570,123.825,-49.894,-178.237,5.688,148.475
C05125=1223.575,123.576,-49.875,-178.240,5.687,148.476
C05126=1223.580,123.327,-49.854,-178.243,5.685,148.476
C05127=1223.584,123.077,-49.834,-178.245,5.685,148.477
C05128=1223.589,122.828,-49.814,-178.247,5.684,148.477
C05129=1223.594,122.579,-49.795,-178.251,5.682,148.478
C05130=1223.599,122.330,-49.775,-178.253,5.681,148.478
C05131=1223.603,122.081,-49.755,-178.255,5.681,148.479
C05132=1223.608,121.831,-49.735,-178.259,5.679,148.480
C05133=1223.613,121.582,-49.716,-178.261,5.678,148.480
C05134=1223.618,121.333,-49.695,-178.263,5.678,148.481
C05135=1223.623,121.084,-49.676,-178.265,5.677,148.481
C05136=1223.628,120.835,-49.657,-178.269,5.675,148.482
C05137=1223.632,120.586,-49.636,-178.271,5.674,148.482
C05138=1223.637,120.336,-49.617,-178.273,5.674,148.483
C05139=1223.642,120.087,-49.597,-178.276,5.672,148.483
C05140=1223.647,119.838,-49.578,-178.279,5.671,148.484
C05141=1223.652,119.589,-49.557,-178.281,5.671,148.484
C05142=1223.656,119.340,-49.538,-178.284,5.669,148.485
C05143=1223.662,119.091,-49.518,-178.286,5.668,148.485
C05144=1223.666,118.841,-49.499,-178.289,5.667,148.486
C05145=1223.670,118.592,-49.479,-178.292,5.666,148.486
C05146=1223.675,118.344,-49.460,-178.294,5.665,148.487
C05147=1223.680,118.094,-49.440,-178.297,5.664,148.488
C05148=1223.685,117.844,-49.420,-178.299,5.663,148.488
C05149=1223.690,117.596,-49.401,-178.302,5.662,148.489
C05150=1223.695,117.346,-49.381,-178.304,5.661,148.489
C05151=1223.699,117.097,-49.361,-178.307,5.660,148.490
C05152=1223.704,116.849,-49.342,-178.310,5.659,148.490
C05153=1223.709,116.599,-49.323,-178.312,5.658,148.491
C05154=1223.714,116.349,-49.303,-178.314,5.657,148.491
C05155=1223.719,116.101,-49.284,-178.317,5.655,148.492
C05156=1223.724,115.851,-49.264,-178.320,5.655,148.492
C05157=1223.728,115.602,-49.245,-178.322,5.654,148.493
C05158=1223.733,115.353,-49.226,-178.324,5.653,148.493
C05159=1223.738,115.103,-49.206,-178.328,5.652,148.494
C05160=1223.742,114.854,-49.186,-178.330,5.651,148.494
C05161=1223.748,114.605,-49.166,-178.332,5.650,148.495
C05162=1223.752,114.356,-49.147,-178.335,5.648,148.495
C05163=1223.757,114.107,-49.128,-178.338,5.648,148.496
C05164=1223.762,113.858,-49.108,-178.340,5.647,148.497
C05165=1223.766,113.608,-49.089,-178.342,5.646,148.497
C05166=1223.772,113.359,-49.069,-178.346,5.645,148.498
C05167=1223.776,113.110,-49.050,-178.348,5.644,148.498
C05168=1223.781,112.861,-49.031,-178.350,5.643,148.499
C05169=1223.786,112.612,-49.011,-178.353,5.643,148.499
C05170=1223.790,112.362,-48.992,-178.356,5.641,148.500
C05171=1223.795,112.113,-48.973,-178.358,5.640,148.500
C05172=1223.800,111.864,-48.953,-178.360,5.639,148.501
C05173=1223.805,111.615,-48.934,-178.364,5.638,148.502
C05174=1223.809,111.366,-48.915,-178.366,5.637,148.502
C05175=1223.815,111.117,-48.896,-178.368,5.636,148.503
C05176=1223.820,110.867,-48.877,-178.371,5.636,148.503
C05177=1223.824,110.617,-48.858,-178.374,5.634,148.504
C05178=1223.829,110.369,-48.838,-178.376,5.633,148.504
C05179=1223.834,110.119,-48.819,-178.379,5.633,148.505
C05180=1223.838,109.870,-48.800,-178.381,5.632,148.505
C05181=1223.843,109.621,-48.780,-178.384,5.630,148.506
C05182=1223.848,109.372,-48.761,-178.386,5.629,148.506
C05183=1223.852,109.123,-48.742,-178.389,5.629,148.507
C05184=1223.858,108.874,-48.723,-178.391,5.628,148.508
C05185=1223.863,108.624,-48.704,-178.394,5.626,148.508
C05186=1223.867,108.375,-48.685,-178.397,5.626,148.509
C05187=1223.872,108.126,-48.665,-178.399,5.625,148.509
C05188=1223.878,107.858,-48.645,-178.401,5.624,148.510
C05189=1223.883,107.588,-48.624,-178.405,5.623,148.510
C05190=1223.888,107.321,-48.604,-178.407,5.622,148.511
C05191=1223.893,107.052,-48.583,-178.410,5.621,148.512
C05192=1223.898,106.803,-48.564,-178.413,5.620,148.512
C05193=1223.902,106.553,-48.545,-178.415,5.619,148.513
C05194=1223.908,106.305,-48.526,-178.418,5.618,148.513
C05195=1223.912,106.055,-48.507,-178.420,5.617,148.514
C05196=1223.917,105.806,-48.488,-178.423,5.616,148.514
C05197=1223.922,105.556,-48.469,-178.426,5.615,148.515
C05198=1223.927,105.308,-48.450,-178.428,5.614,148.515
C05199=1223.931,105.058,-48.431,-178.431,5.613,148.516
C05200=1223.936,104.809,-48.413,-178.433,5.612,148.517
C05201=1223.941,104.559,-48.393,-178.436,5.611,148.517
C05202=1223.946,104.311,-48.374,-178.438,5.611,148.518
C05203=1223.951,104.061,-48.355,-178.440,5.610,148.518
C05204=1223.955,103.812,-48.337,-178.444,5.608,148.519
C05205=1223.960,103.562,-48.317,-178.446,5.608,148.519
C05206=1223.965,103.313,-48.299,-178.448,5.607,148.520
C05207=1223.970,103.064,-48.280,-178.451,5.606,148.521
C05208=1223.974,102.815,-48.261,-178.454,5.605,148.521
C05209=1223.980,102.566,-48.242,-178.456,5.604,148.522
C05210=1223.984,102.316,-48.223,-178.459,5.603,148.522
C05211=1223.989,102.068,-48.204,-178.461,5.602,148.523
C05212=1223.994,101.818,-48.185,-178.464,5.602,148.523
C05213=1223.999,101.569,-48.166,-178.467,5.600,148.524
C05214=1224.004,101.320,-48.148,-178.469,5.599,148.524
C05215=1224.009,101.070,-48.128,-178.472,5.599,148.525
C05216=1224.013,100.821,-48.110,-178.474,5.598,148.526
C05217=1224.017,100.572,-48.091,-178.476,5.597,148.526
C05218=1224.023,100.322,-48.073,-178.480,5.596,148.527
C05219=1224.028,100.074,-48.054,-178.482,5.595,148.527
C05220=1224.032,99.824,-48.034,-178.484,5.594,148.528
C05221=1224.037,99.575,-48.016,-178.487,5.594,148.528
C05222=1224.041,99.326,-47.997,-178.490,5.593,148.529
C05223=1224.047,99.076,-47.979,-178.492,5.591,148.529
C05224=1224.052,98.828,-47.960,-178.495,5.591,148.530
C05225=1224.057,98.577,-47.941,-178.497,5.590,148.531
C05226=1224.062,98.328,-47.923,-178.500,5.589,148.531
C05227=1224.066,98.080,-47.904,-178.502,5.588,148.532
C05228=1224.071,97.829,-47.886,-178.505,5.587,148.532
C05229=1224.076,97.581,-47.867,-178.508,5.586,148.533
C05230=1224.081,97.332,-47.849,-178.510,5.585,148.534
C05231=1224.086,97.082,-47.829,-178.513,5.585,148.534
C05232=1224.090,96.833,-47.811,-178.515,5.584,148.535
C05233=1224.095,96.584,-47.793,-178.518,5.582,148.535
C05234=1224.100,96.334,-47.774,-178.521,5.582,148.536
C05235=1224.105,96.085,-47.756,-178.523,5.581,148.536
C05236=1224.110,95.836,-47.737,-178.525,5.580,148.537
C05237=1224.115,95.586,-47.718,-178.528,5.580,148.538
C05238=1224.120,95.337,-47.700,-178.530,5.579,148.538
C05239=1224.124,95.089,-47.681,-178.533,5.577,148.539
C05240=1224.129,94.838,-47.662,-178.536,5.577,148.539
C05241=1224.134,94.589,-47.644,-178.538,5.576,148.540
C05242=1224.139,94.341,-47.626,-178.541,5.575,148.540
C05243=1224.143,94.091,-47.607,-178.543,5.575,148.541
C05244=1224.149,93.841,-47.589,-178.545,5.574,148.541
C05245=1224.153,93.593,-47.570,-178.549,5.572,148.542
C05246=1224.158,93.344,-47.552,-178.551,5.572,148.543
C05247=1224.163,93.094,-47.534,-178.553,5.571,148.543
C05248=1224.168,92.845,-47.514,-178.556,5.570,148.544
C05249=1224.173,92.596,-47.496,-178.559,5.569,148.544
C05250=1224.178,92.346,-47.479,-178.561,5.569,148.545
C05251=1224.182,92.097,-47.460,-178.564,5.567,148.546
C05252=1224.187,91.848,-47.441,-178.567,5.566,148.546
C05253=1224.192,91.599,-47.423,-178.569,5.566,148.547
C05254=1224.197,91.349,-47.405,-178.571,5.565,148.547
C05255=1224.201,91.099,-47.387,-178.574,5.564,148.548
C05256=1224.206,90.850,-47.369,-178.577,5.564,148.549
C05257=1224.212,90.601,-47.349,-178.579,5.563,148.549
C05258=1224.217,90.352,-47.331,-178.582,5.561,148.550
C05259=1224.221,90.102,-47.313,-178.585,5.561,148.550
C05260=1224.226,89.853,-47.295,-178.587,5.560,148.551
C05261=1224.231,89.604,-47.277,-178.589,5.559,148.551
C05262=1224.236,89.355,-47.259,-178.592,5.559,148.552
C05263=1224.240,89.106,-47.240,-178.595,5.558,148.553
C05264=1224.245,88.856,-47.221,-178.597,5.557,148.553
C05265=1224.250,88.607,-47.203,-178.600,5.556,148.554
C05266=1224.255,88.358,-47.185,-178.602,5.555,148.554
C05267=1224.260,88.109,-47.167,-178.605,5.554,148.555
C05268=1224.264,87.859,-47.149,-178.607,5.553,148.555
C05269=1224.269,87.610,-47.131,-178.610,5.553,148.556
C05270=1224.274,87.360,-47.113,-178.612,5.552,148.557
C05271=1224.279,87.111,-47.095,-178.615,5.551,148.557
C05272=1224.285,86.862,-47.077,-178.618,5.550,148.558
C05273=1224.290,86.613,-47.059,-178.620,5.549,148.558
C05274=1224.294,86.363,-47.040,-178.623,5.549,148.559
C05275=1224.299,86.113,-47.022,-178.625,5.548,148.560
C05276=1224.304,85.864,-47.004,-178.628,5.547,148.560
C05277=1224.308,85.616,-46.986,-178.630,5.547,148.561
C05278=1224.313,85.367,-46.968,-178.633,5.546,148.561
C05279=1224.318,85.117,-46.950,-178.635,5.545,148.562
C05280=1224.323,84.867,-46.932,-178.638,5.544,148.563
C05281=1224.328,84.618,-46.914,-178.641,5.543,148.563
C05282=1224.333,84.369,-46.896,-178.643,5.542,148.564
C05283=1224.338,84.119,-46.878,-178.646,5.541,148.564
C05284=1224.343,83.870,-46.860,-178.648,5.541,148.565
C05285=1224.347,83.621,-46.842,-178.650,5.540,148.565
C05286=1224.352,83.372,-46.824,-178.653,5.539,148.566
C05287=1224.357,83.122,-46.806,-178.656,5.539,148.567
C05288=1224.362,82.873,-46.788,-178.658,5.538,148.567
C05289=1224.366,82.624,-46.770,-178.661,5.536,148.568
C05290=1224.371,82.374,-46.752,-178.664,5.536,148.568
C05291=1224.376,82.125,-46.734,-178.666,5.535,148.569
C05292=1224.381,81.857,-46.714,-178.669,5.535,148.570
C05293=1224.387,81.588,-46.696,-178.672,5.534,148.570
C05294=1224.392,81.320,-46.676,-178.675,5.533,148.571
C05295=1224.397,81.052,-46.657,-178.677,5.532,148.572
C05296=1224.402,80.802,-46.639,-178.679,5.531,148.572
C05297=1224.407,80.553,-46.621,-178.682,5.530,148.573
C05298=1224.412,80.303,-46.604,-178.685,5.530,148.573
C05299=1224.417,80.054,-46.586,-178.687,5.529,148.574
C05300=1224.422,79.805,-46.568,-178.689,5.528,148.575
C05301=1224.427,79.556,-46.550,-178.692,5.528,148.575
C05302=1224.432,79.307,-46.532,-178.695,5.527,148.576
C05303=1224.437,79.057,-46.515,-178.698,5.526,148.577
C05304=1224.442,78.808,-46.497,-178.700,5.525,148.577
C05305=1224.447,78.559,-46.479,-178.703,5.524,148.578
C05306=1224.451,78.310,-46.461,-178.705,5.524,148.578
C05307=1224.455,78.059,-46.444,-178.708,5.523,148.579
C05308=1224.460,77.810,-46.426,-178.710,5.522,148.579
C05309=1224.465,77.561,-46.408,-178.713,5.522,148.580
C05310=1224.470,77.312,-46.390,-178.715,5.521,148.581
C05311=1224.475,77.062,-46.372,-178.718,5.520,148.581
C05312=1224.480,76.813,-46.354,-178.721,5.520,148.582
C05313=1224.485,76.564,-46.337,-178.723,5.519,148.582
C05314=1224.490,76.314,-46.320,-178.725,5.518,148.583
C05315=1224.495,76.065,-46.302,-178.729,5.517,148.584
C05316=1224.500,75.816,-46.284,-178.731,5.516,148.584
C05317=1224.505,75.566,-46.267,-178.733,5.515,148.585
C05318=1224.510,75.317,-46.249,-178.736,5.515,148.585
C05319=1224.514,75.068,-46.231,-178.739,5.514,148.586
C05320=1224.519,74.818,-46.214,-178.741,5.514,148.587
C05321=1224.524,74.569,-46.196,-178.743,5.513,148.587
C05322=1224.529,74.320,-46.178,-178.746,5.512,148.588
C05323=1224.533,74.070,-46.161,-178.749,5.511,148.589
C05324=1224.538,73.821,-46.143,-178.751,5.511,148.589
C05325=1224.544,73.571,-46.126,-178.753,5.510,148.590
C05326=1224.548,73.322,-46.108,-178.756,5.509,148.590
C05327=1224.554,73.072,-46.091,-178.759,5.509,148.591
C05328=1224.558,72.824,-46.074,-178.761,5.508,148.592
C05329=1224.563,72.575,-46.056,-178.764,5.508,148.592
C05330=1224.569,72.325,-46.039,-178.766,5.507,148.593
C05331=1224.573,72.076,-46.021,-178.769,5.505,148.593
C05332=1224.578,71.827,-46.004,-178.772,5.505,148.594
C05333=1224.583,71.577,-45.986,-178.774,5.504,148.595
C05334=1224.588,71.328,-45.969,-178.777,5.504,148.595
C05335=1224.592,71.079,-45.951,-178.779,5.503,148.596
C05336=1224.597,70.829,-45.934,-178.782,5.502,148.596
C05337=1224.602,70.580,-45.916,-178.784,5.501,148.597
C05338=1224.607,70.330,-45.899,-178.787,5.501,148.598
C05339=1224.612,70.081,-45.881,-178.789,5.500,148.598
C05340=1224.617,69.831,-45.864,-178.792,5.499,148.599
C05341=1224.621,69.582,-45.847,-178.795,5.499,148.599
C05342=1224.626,69.333,-45.829,-178.797,5.498,148.600
C05343=1224.632,69.084,-45.812,-178.800,5.498,148.601
C05344=1224.636,68.835,-45.795,-178.802,5.497,148.601
C05345=1224.642,68.585,-45.778,-178.805,5.496,148.602
C05346=1224.646,68.336,-45.760,-178.807,5.495,148.603
C05347=1224.651,68.086,-45.743,-178.810,5.495,148.603
C05348=1224.656,67.837,-45.725,-178.812,5.494,148.604
C05349=1224.661,67.587,-45.708,-178.815,5.493,148.604
C05350=1224.666,67.338,-45.691,-178.817,5.493,148.605
C05351=1224.670,67.089,-45.673,-178.820,5.492,148.606
C05352=1224.676,66.840,-45.657,-178.822,5.492,148.606
C05353=1224.681,66.590,-45.640,-178.825,5.491,148.607
C05354=1224.686,66.341,-45.622,-178.827,5.490,148.607
C05355=1224.690,66.091,-45.605,-178.830,5.490,148.608
C05356=1224.695,65.842,-45.588,-178.832,5.489,148.609
C05357=1224.700,65.593,-45.570,-178.836,5.488,148.609
C05358=1224.705,65.343,-45.553,-178.838,5.487,148.610
C05359=1224.710,65.094,-45.537,-178.840,5.486,148.610
C05360=1224.715,64.845,-45.519,-178.843,5.486,148.611
C05361=1224.720,64.595,-45.502,-178.846,5.485,148.612
C05362=1224.724,64.346,-45.485,-178.848,5.484,148.612
C05363=1224.730,64.096,-45.468,-178.851,5.484,148.613
C05364=1224.734,63.847,-45.450,-178.853,5.483,148.614
C05365=1224.740,63.598,-45.433,-178.856,5.482,148.614
C05366=1224.744,63.348,-45.417,-178.858,5.482,148.615
C05367=1224.749,63.099,-45.400,-178.861,5.481,148.616
C05368=1224.754,62.850,-45.382,-178.864,5.481,148.616
C05369=1224.759,62.600,-45.365,-178.866,5.480,148.617
C05370=1224.764,62.351,-45.349,-178.868,5.479,148.617
C05371=1224.769,62.101,-45.331,-178.871,5.478,148.618
C05372=1224.774,61.852,-45.315,-178.874,5.478,148.619
C05373=1224.778,61.603,-45.297,-178.876,5.477,148.619
C05374=1224.783,61.353,-45.280,-178.879,5.477,148.620
C05375=1224.789,61.104,-45.263,-178.881,5.476,148.620
C05376=1224.793,60.855,-45.246,-178.884,5.475,148.621
C05377=1224.798,60.605,-45.229,-178.886,5.475,148.622
C05378=1224.803,60.355,-45.212,-178.889,5.474,148.622
C05379=1224.808,60.107,-45.195,-178.892,5.474,148.623
C05380=1224.813,59.857,-45.178,-178.894,5.473,148.624
C05381=1224.817,59.608,-45.162,-178.896,5.472,148.624
C05382=1224.823,59.358,-45.144,-178.899,5.471,148.625
C05383=1224.828,59.109,-45.128,-178.902,5.471,148.626
C05384=1224.833,58.860,-45.111,-178.904,5.470,148.626
C05385=1224.837,58.610,-45.094,-178.907,5.470,148.627
C05386=1224.842,58.361,-45.077,-178.910,5.469,148.628
C05387=1224.848,58.112,-45.060,-178.912,5.468,148.628
C05388=1224.852,57.862,-45.044,-178.914,5.468,148.629
C05389=1224.857,57.612,-45.027,-178.917,5.467,148.629
C05390=1224.862,57.363,-45.010,-178.920,5.467,148.630
C05391=1224.867,57.114,-44.994,-178.922,5.466,148.631
C05392=1224.872,56.864,-44.976,-178.925,5.465,148.631
C05393=1224.877,56.615,-44.960,-178.926,5.465,148.632
C05394=1224.882,56.366,-44.943,-178.929,5.465,148.632
C05395=1224.887,56.116,-44.926,-178.932,5.464,148.633
C05396=1224.892,55.848,-44.908,-178.935,5.463,148.634
C05397=1224.898,55.579,-44.890,-178.938,5.462,148.634
C05398=1224.902,55.311,-44.872,-178.940,5.462,148.635
C05399=1224.908,55.043,-44.854,-178.943,5.461,148.636
C05400=1224.913,54.793,-44.837,-178.945,5.460,148.636
C05401=1224.918,54.544,-44.820,-178.948,5.460,148.637
C05402=1224.923,54.294,-44.804,-178.951,5.459,148.638
C05403=1224.928,54.044,-44.787,-178.953,5.459,148.638
C05404=1224.933,53.796,-44.771,-178.956,5.458,148.639
C05405=1224.937,53.546,-44.754,-178.958,5.457,148.639
C05406=1224.943,53.296,-44.737,-178.961,5.457,148.640
C05407=1224.948,53.048,-44.720,-178.963,5.456,148.641
C05408=1224.952,52.798,-44.704,-178.966,5.456,148.641
C05409=1224.957,52.549,-44.687,-178.969,5.455,148.642
C05410=1224.962,52.300,-44.670,-178.971,5.454,148.643
C05411=1224.967,52.049,-44.654,-178.973,5.455,148.644
C05412=1224.972,51.800,-44.638,-178.976,5.454,148.644
C05413=1224.977,51.551,-44.621,-178.978,5.453,148.645
C05414=1224.982,51.301,-44.604,-178.981,5.453,148.645
C05415=1224.987,51.053,-44.588,-178.983,5.452,148.646
C05416=1224.992,50.803,-44.571,-178.986,5.451,148.647
C05417=1224.996,50.553,-44.555,-178.989,5.451,148.647
C05418=1225.001,50.304,-44.539,-178.991,5.450,148.648
C05419=1225.007,50.054,-44.522,-178.993,5.449,148.648
C05420=1225.011,49.805,-44.505,-178.996,5.449,148.649
C05421=1225.016,49.556,-44.489,-178.999,5.448,148.650
C05422=1225.021,49.306,-44.473,-179.001,5.448,148.650
C05423=1225.026,49.057,-44.456,-179.004,5.447,148.651
C05424=1225.031,48.807,-44.439,-179.007,5.447,148.652
C05425=1225.036,48.558,-44.422,-179.009,5.446,148.652
C05426=1225.041,48.309,-44.407,-179.012,5.445,148.653
C05427=1225.046,48.059,-44.390,-179.014,5.445,148.654
C05428=1225.051,47.810,-44.374,-179.017,5.444,148.654
C05429=1225.056,47.560,-44.358,-179.019,5.443,148.655
C05430=1225.061,47.311,-44.342,-179.021,5.444,148.656
C05431=1225.066,47.062,-44.324,-179.024,5.443,148.656
C05432=1225.070,46.812,-44.308,-179.027,5.443,148.657
C05433=1225.076,46.563,-44.292,-179.029,5.442,148.658
C05434=1225.080,46.313,-44.275,-179.032,5.441,148.658
C05435=1225.085,46.065,-44.259,-179.034,5.441,148.659
C05436=1225.090,45.814,-44.243,-179.037,5.440,148.659
C05437=1225.095,45.566,-44.227,-179.039,5.439,148.660
C05438=1225.100,45.316,-44.211,-179.042,5.439,148.661
C05439=1225.106,45.066,-44.194,-179.045,5.438,148.661
C05440=1225.110,44.817,-44.177,-179.047,5.438,148.662
C05441=1225.116,44.568,-44.162,-179.050,5.437,148.663
C05442=1225.120,44.318,-44.145,-179.053,5.437,148.663
C05443=1225.125,44.069,-44.129,-179.055,5.436,148.664
C05444=1225.130,43.819,-44.113,-179.057,5.436,148.665
C05445=1225.134,43.570,-44.096,-179.059,5.435,148.665
C05446=1225.140,43.320,-44.081,-179.062,5.435,148.666
C05447=1225.144,43.071,-44.064,-179.065,5.434,148.667
C05448=1225.150,42.821,-44.048,-179.067,5.434,148.667
C05449=1225.154,42.572,-44.032,-179.070,5.433,148.668
C05450=1225.160,42.323,-44.016,-179.073,5.433,148.669
C05451=1225.165,42.074,-44.000,-179.075,5.432,148.669
C05452=1225.169,41.824,-43.984,-179.077,5.431,148.670
C05453=1225.174,41.575,-43.967,-179.080,5.431,148.670
C05454=1225.179,41.325,-43.951,-179.083,5.430,148.671
C05455=1225.184,41.076,-43.935,-179.085,5.430,148.672
C05456=1225.189,40.826,-43.919,-179.087,5.430,148.672
C05457=1225.194,40.577,-43.903,-179.090,5.429,148.673
C05458=1225.199,40.327,-43.887,-179.093,5.429,148.674
C05459=1225.204,40.078,-43.871,-179.095,5.428,148.674
C05460=1225.209,39.828,-43.855,-179.098,5.427,148.675
C05461=1225.214,39.579,-43.838,-179.100,5.427,148.675
C05462=1225.219,39.329,-43.822,-179.103,5.426,148.676
C05463=1225.224,39.080,-43.807,-179.105,5.425,148.677
C05464=1225.229,38.831,-43.791,-179.108,5.425,148.678
C05465=1225.234,38.581,-43.775,-179.110,5.425,148.678
C05466=1225.239,38.332,-43.758,-179.113,5.425,148.679
C05467=1225.244,38.082,-43.742,-179.115,5.424,148.680
C05468=1225.249,37.833,-43.727,-179.118,5.423,148.680
C05469=1225.254,37.583,-43.710,-179.121,5.423,148.681
C05470=1225.259,37.334,-43.695,-179.123,5.422,148.682
C05471=1225.263,37.085,-43.679,-179.125,5.421,148.682
C05472=1225.268,36.835,-43.663,-179.128,5.421,148.683
C05473=1225.274,36.586,-43.647,-179.131,5.420,148.683
